# B&R Automation Studio project AAU12Segmenter (part 9)

#### mxA_Main.st - not listed in the package file held
```iecst
PROGRAM _INIT

	FOR i:=0 TO 5 DO
		KUKAs[i].AxisGroupIdx := i + 1;
		KUKAs[i].gripperAction.whitePin := ADR(gripperWhitePins[i]);
		KUKAs[i].gripperAction.blackPin := ADR(gripperBlackPins[i]);
		KUKAs[i].gripperAction.action := OPEN;
		KUKAs[i].gripperAction();
		KUKAs[i].cm.state := 0;
		KUKAs[i].startState := 0;
	END_FOR

	KUKAs[0].eeType := COVER_EE;
	KUKAs[1].eeType := DRILL_EE;
	KUKAs[2].eeType := PCB_EE;
	KUKAs[3].eeType := FUSE_EE;
	KUKAs[4].eeType := COVER_EE;
	KUKAs[5].eeType := COVER_EE;

END_PROGRAM

PROGRAM _CYCLIC

	// Loop through each robot for configurations
	FOR i := 0 TO 5 DO

		////////// Temporary skip until problem with library for Kuka KR4 is solved///////////
		IF i = 0 OR i = 5 THEN

			RETURN;

		END_IF

		/////////////////////////////////////////////////////
		// Logic to transform USINT (Input) to BYTE (FUBS) //
		/////////////////////////////////////////////////////

		brsmemcpy(ADR(KRC_Input[0]),ADR(InputVariables[i,0]), 254);

		/////////////////////////////////////////////////////
		// KRC_ReadAxisGroup has to be called at the Begin //
		// of the Cyclic Task to get all the Information   //
		// From the KRC from all KUKAs					   //
		/////////////////////////////////////////////////////

		KUKAs[i].start.KRC_ReadAxisGroup.KRC4_Input 			:= ADR(KRC_Input);
		KUKAs[i].start.KRC_ReadAxisGroup.AxisGroupIdx 			:= KUKAs[i].AxisGroupIdx;
		KUKAs[i].start.KRC_ReadAxisGroup.KRC_AxisGroupRefArr 	:= ADR(AxisRef);

		KUKAs[i].start.KRC_ReadAxisGroup();

		/////////////////////////////////////////////////////
		// Call User functions                             //
		/////////////////////////////////////////////////////

		pKuka ACCESS ADR(KUKAs[i]);
		cm ACCESS ADR(KUKAs[i].cm);

		// mxA_Start contains FB calls associated with initialization of the robots and diagnosis
		mxA_Start;

		//mxA_JointMovement;
		//mxA_LinearMovement;
		//mxA_ErrorMessage;

		CASE i OF
			1:
				mxA_KUKA1;

			2:
				mxA_KUKA2;

			3:
				mxA_KUKA3;

			4:
				mxA_KUKA4;

			5:
				mxA_KUKA5;

			6:
				mxA_KUKA6;

		END_CASE

		//mxA_KUKA6;

		/////////////////////////////////////////////////////
		// FunctionBlock to write the Output on the Struct //
		/////////////////////////////////////////////////////

		KUKAs[i].start.KRC_WriteAxisGroup.AxisGroupIdx			:= KUKAs[i].AxisGroupIdx;
		KUKAs[i].start.KRC_WriteAxisGroup.KRC_AxisGroupRefArr 	:= ADR(AxisRef);
		KUKAs[i].start.KRC_WriteAxisGroup.KRC4_Output 			:= ADR(KRC_Output);

		KUKAs[i].start.KRC_WriteAxisGroup();

		/////////////////////////////////////////////////////
		// Logic to transform BYTE (FUBS) to USINT (Input) //
		/////////////////////////////////////////////////////
		brsmemcpy(ADR(OutputVariables[i,0]),ADR(KRC_Output[0]), 254);

	END_FOR

END_PROGRAM
```

#### mxA_Start.st - not listed in the package file held
```iecst
ACTION mxA_Start:

	CASE pKuka.startState OF

		0: // Configuring KUKA FBs once

			// Logic to call the KRC_Initialize
			pKuka.start.KRC_Initialize.AxisGroupIdx 				:= pKuka.AxisGroupIdx;
			pKuka.start.KRC_Initialize.KRC_AxisGroupRefArr 			:= ADR(AxisRef);

			// Logic to call the KRC_Error
			pKuka.start.KRC_Error.AxisGroupIdx 						:= pKuka.AxisGroupIdx;
			pKuka.start.KRC_Error.MessageReset 						:= FALSE; // REMEMBER TO CHANGE LATER
			pKuka.start.KRC_Error.KRC_AxisGroupRefArr				:= ADR(AxisRef);

			// Logic to call KRC_AutomaticExternal
			pKuka.start.KRC_AutomaticExternal.AxisGroupIdx 			:= pKuka.AxisGroupIdx;
			pKuka.start.KRC_AutomaticExternal.MOVE_ENABLE 			:= TRUE;
			pKuka.start.KRC_AutomaticExternal.DRIVES_OFF 			:= TRUE;
			pKuka.start.KRC_AutomaticExternal.KRC_AxisGroupRefArr	:= ADR(AxisRef);
			pKuka.start.KRC_AutomaticExternal.EXT_START 			:= FALSE; // Binded to Continue Prog in original program
			pKuka.start.KRC_AutomaticExternal.ENABLE_T1 			:= TRUE;
			pKuka.start.KRC_AutomaticExternal.ENABLE_EXT 			:= TRUE;

			// Logic for startup of robot
			pKuka.start.KRC_AutoStart.AxisGroupIdx 					:= pKuka.AxisGroupIdx;
			pKuka.start.KRC_AutoStart.KRC_AxisGroupRefArr 			:= ADR(AxisRef);
			pKuka.start.KRC_AutoStart.ExecuteReset 					:= FALSE; // REMEMBER TO CHANGE LATER

			// Logic to set override for robot velocity
			pKuka.start.KRC_SetOverride.AxisGroupIdx 				:= pKuka.AxisGroupIdx;
			pKuka.start.KRC_SetOverride.KRC_AxisGroupRefArr 		:= ADR(AxisRef);
			pKuka.start.KRC_SetOverride.Override 					:= 10; // REMEMBER TO CHANGE LATER

			// Logic to set
			pKuka.start.KRC_Abort.AxisGroupIdx 						:= pKuka.AxisGroupIdx;
			pKuka.start.KRC_Abort.KRC_AxisGroupRefArr				:= ADR(AxisRef);
			pKuka.start.KRC_Abort.ExecuteCmd						:= FALSE;  /// Used to be set by HMI - Remember to incorporate it later

			// Logic to set KRC_Diag
			pKuka.start.KRC_Diag.AxisGroupIdx 						:= pKuka.AxisGroupIdx;
			pKuka.start.KRC_Diag.KRC_AxisGroupRefArr 				:= ADR(AxisRef);
			pKuka.start.KRC_Diag.ShowTrace 							:= FALSE;

			pKuka.startState  := 1;

		1: // Wait for P, S and EXT
			IF pKuka.status.P_ AND pKuka.status.S_ AND pKuka.status.EXT_ THEN

				pKuka.startState  := 2;

			END_IF

		2: // Reset KRC errors and autostart
			pKuka.start.KRC_Error.MessageReset := TRUE;
			pKuka.start.KRC_AutoStart.ExecuteReset := TRUE;

			IF pKuka.status.R_ AND pKuka.status.I_ THEN

				pKuka.start.KRC_Error.MessageReset := FALSE;
				pKuka.start.KRC_AutoStart.ExecuteReset := FALSE;
				pKuka.startState  := 3;

			END_IF

		3: // Check if any error occurred
			IF 	NOT pKuka.status.P_ OR
				NOT pKuka.status.S_ OR
				NOT pKuka.status.EXT_ OR
				NOT pKuka.status.R_ OR
				NOT pKuka.status.I_ THEN

				pKuka.startState  := 1;

			END_IF

	END_CASE

	// Logic to call the KRC_Initialize
	// KRC_Initialize gives back the Status OF the like, online, Initialized,.......
	pKuka.start.KRC_Initialize();

	// Logic to call the KRC_Error.
	// KRC_Error gives back the Status OF the Robot like, online, Initialized,.......
	pKuka.start.KRC_Error();

	// KRC_AutomaticExternal allows to control the Robot with the PLC
	pKuka.start.KRC_AutomaticExternal();

	//Function Block for StartUp of Robot
	pKuka.start.KRC_AutoStart();

	// KRC_SetOverride used to set the Override for the Robot Velocity
	pKuka.start.KRC_SetOverride();

	// KRC_Abort cancels all active and buffered statements and motions
	pKuka.start.KRC_Abort();

	// KRC_Diag gives back some information about the axis and robot
	pKuka.start.KRC_Diag();

	//Checking status of KRC and PLC for creating the signals for the HMI
	IF pKuka.start.KRC_Diag.ProconosCyc_Act = -1 OR pKuka.start.KRC_Error.NoHeartbeatPCOS THEN
		pKuka.status.P_ := FALSE;
	ELSE
		pKuka.status.P_ := TRUE;
	END_IF

	IF pKuka.start.KRC_Diag.SubmitCyc_Act = -1 OR pKuka.start.KRC_Error.NoHeartbeatKRC THEN
		pKuka.status.S_ := FALSE;
	ELSE
		pKuka.status.S_ := TRUE;
	END_IF

	IF pKuka.start.KRC_AutomaticExternal.EXT THEN
		pKuka.status.EXT_ := TRUE;
	ELSE
		pKuka.status.EXT_ := FALSE;
	END_IF

	IF NOT pKuka.start.KRC_Error.DrivesNotReady AND pKuka.start.KRC_AutomaticExternal.RC_RDY1 THEN
		pKuka.status.I_ := TRUE;
	ELSE
		pKuka.status.I_ := FALSE;
	END_IF

	IF pKuka.start.KRC_AutoStart.DispActive THEN
		pKuka.status.R_	:= TRUE;
	ELSE
		pKuka.status.R_	:= FALSE;
	END_IF

END_ACTION
```

#### RobotHandling.st - not listed in the package file held
```iecst
ACTION RobotHandling:
	CASE cm.state OF

		1000:
			IF robotExecute[i] THEN
				cm.description := 'Move to pickup point with relative linear movement';
				robotBusy[i] := TRUE;
				pKuka.convert.ValuesToCOORDSYS.IPO_Mode := 1; // #TOOL
				pKuka.convert.ValuesToCOORDSYS();

				pKuka.motion.KRC_MoveLinearRelative.CoordinateSystem := pKuka.convert.ValuesToCOORDSYS.COORDSYS;

				pKuka.tempPosition.X := pKuka.tempPosition.Y := pKuka.tempPosition.Z := pKuka.tempPosition.A := pKuka.tempPosition.B := pKuka.tempPosition.C
				:= 0;
				pKuka.tempPosition.Z := -relativeDistance;
				// Status and turn is already set from moving to approach point

				pKuka.motion.KRC_MoveLinearRelative.Position := pKuka.tempPosition;

				pKuka.motion.KRC_MoveLinearRelative.ExecuteCmd := TRUE;
				IF pKuka.motion.KRC_MoveLinearRelative.Done THEN
					pKuka.motion.KRC_MoveLinearRelative.ExecuteCmd := FALSE;
					cm.state := 1010;
				END_IF
			END_IF

		1010:
			cm.description := 'Close gripper and wait a little before moving to ensure proper grip';

			pKuka.gripperAction.action := CLOSE;

			pKuka.TON.PT := REAL_TO_TIME(gripperWaitTime); // in ms
			pKuka.TON.IN := TRUE;
			IF pKuka.TON.Q THEN
				pKuka.TON.IN := FALSE;
				cm.state := 1020;
			END_IF

		1020:
			cm.description := 'Move back to approach point with relative linear movement';

			pKuka.tempPosition.X := pKuka.tempPosition.Y := pKuka.tempPosition.Z := pKuka.tempPosition.A := pKuka.tempPosition.B := pKuka.tempPosition.C
			:= 0;
			pKuka.tempPosition.Z := relativeDistance;
			// Status and turn is already set from moving to approach point

			pKuka.motion.KRC_MoveLinearRelative.Position := pKuka.tempPosition;

			pKuka.motion.KRC_MoveLinearRelative.ExecuteCmd := TRUE;
			IF pKuka.motion.KRC_MoveLinearRelative.Done THEN
				pKuka.motion.KRC_MoveLinearRelative.ExecuteCmd := FALSE;
				cm.state := 1030;
			END_IF

		1030:
			cm.description := 'Move to approach point of magazine with absolute direct movement';

			pKuka.convert.ValuesToPosition.posType := APPROACH_MAGAZINE;
			pKuka.convert.ValuesToPosition();

			pKuka.convert.ValuesToCOORDSYS.Base := pKuka.convert.ValuesToPosition.baseNo; // Magazine frame
			pKuka.convert.ValuesToCOORDSYS.IPO_Mode := 0; // #BASE
			pKuka.convert.ValuesToCOORDSYS();

			pKuka.tempPosition := pKuka.convert.ValuesToPosition.outputPos;

			pKuka.motion.KRC_MoveDirectAbsolute.CoordinateSystem := pKuka.convert.ValuesToCOORDSYS.COORDSYS;
			pKuka.motion.KRC_MoveDirectAbsolute.Position := pKuka.tempPosition;

			pKuka.motion.KRC_MoveDirectAbsolute.ExecuteCmd := TRUE;
			IF pKuka.motion.KRC_MoveDirectAbsolute.Done THEN
				pKuka.motion.KRC_MoveDirectAbsolute.ExecuteCmd := FALSE;
				cm.state := 1040;
			END_IF

		1040:
			cm.description := 'Define order-specific approach point at magazine';

			pKuka.convert.ValuesToPosition.posType := APPROACH_MAGAZINE;
			pKuka.convert.ValuesToPosition();

			pKuka.tempPosition := pKuka.convert.ValuesToPosition.outputPos;

			CASE pKuka.axisGroupIdx OF
				6:
					// Determine the stack the manipulator should go to depending on the ID of the order
					FOR k := 0 TO (unloadSizeX*unloadSizeY - 1) DO
						xIdxTemp := k MOD unloadSizeX;
						yIdxTemp := REAL_TO_INT(brmfloor(k / unloadSizeX));

						// If the ID already has a stack
						IF idAtStack[xIdxTemp, yIdxTemp] = orderSpec[i] THEN
							// If an non-taken stack was selected, reset it
							IF (xIdx <> -1 OR yIdx <> -1) THEN
								idAtStack[xIdx, yIdx] := -1;
							END_IF
							xIdx := xIdxTemp;
							yIdx := yIdxTemp;
							EXIT;
						END_IF

						IF (xIdx = -1 OR yIdx = -1) AND (idAtStack[xIdxTemp, yIdxTemp] = -1 AND stackCounter[xIdxTemp, yIdxTemp] + orderAmount <= unloadSizeZ) THEN
							xIdx := xIdxTemp;
							yIdx := yIdxTemp;
							idAtStack[xIdx, yIdx] := orderSpec[i];
						END_IF

					END_FOR

					// Determine the position from x- and y-index
					pKuka.tempPosition.X := pKuka.tempPosition.X + xIdx * 120;
					pKuka.tempPosition.Y := pKuka.tempPosition.Y - yIdx * 80;

					// Reset parameters and increment counters
					orderCounter[xIdx, yIdx] := orderCounter[xIdx, yIdx] + 1;
					stackCounter[xIdx, yIdx] := stackCounter[xIdx, yIdx] + 1;
					IF orderCounter[xIdx, yIdx] = orderAmount THEN
						idAtStack[xIdx, yIdx] := -1;
						orderCounter[xIdx, yIdx] := 0;
					END_IF
					xIdx := yIdx := -1;

			END_CASE

			cm.state := 1050;

		1050:
			cm.description := 'Move to order-specific approach point at magazine';
			pKuka.convert.ValuesToCOORDSYS.IPO_Mode := 0; // #BASE
			pKuka.convert.ValuesToCOORDSYS();

			pKuka.motion.KRC_MoveDirectAbsolute.CoordinateSystem := pKuka.convert.ValuesToCOORDSYS.COORDSYS;

			pKuka.motion.KRC_MoveDirectAbsolute.Position := pKuka.tempPosition;

			pKuka.motion.KRC_MoveDirectAbsolute.ExecuteCmd := TRUE;
			IF pKuka.motion.KRC_MoveDirectAbsolute.Done THEN
				pKuka.motion.KRC_MoveDirectAbsolute.ExecuteCmd := FALSE;
				cm.state := 1060;
			END_IF

		1060:
			cm.description := 'Move to place point at magazine with relative movement';

			pKuka.convert.ValuesToCOORDSYS.IPO_Mode := 1; // #TOOL
			pKuka.convert.ValuesToCOORDSYS();

			pKuka.motion.KRC_MoveLinearRelative.CoordinateSystem := pKuka.convert.ValuesToCOORDSYS.COORDSYS;

			pKuka.tempPosition.X := pKuka.tempPosition.Y := pKuka.tempPosition.A := pKuka.tempPosition.B := pKuka.tempPosition.C
			:= 0;
			pKuka.tempPosition.Z := -(pKuka.tempPosition.Z - (unloadSizeZ - stackCounter[xIdx,yIdx])* 21);
			// Status and turn is already set from moving to approach point

			pKuka.motion.KRC_MoveLinearRelative.Position := pKuka.tempPosition;

			pKuka.motion.KRC_MoveLinearRelative.ExecuteCmd := TRUE;
			IF pKuka.motion.KRC_MoveLinearRelative.Done THEN
				pKuka.motion.KRC_MoveLinearRelative.ExecuteCmd := FALSE;
				cm.state := 1070;
			END_IF

		1070:
			cm.description := 'Open gripper and wait a little before moving to ensure proper grip';

			pKuka.gripperAction.action := OPEN;

			pKuka.TON.PT := REAL_TO_TIME(gripperWaitTime); // in ms
			pKuka.TON.IN := TRUE;
			IF pKuka.TON.Q THEN
				pKuka.TON.IN := FALSE;
				cm.state := 1080;
			END_IF

		1080:
			cm.description := 'Move to place point at magazine with relative movement';

			pKuka.convert.ValuesToCOORDSYS.IPO_Mode := 1; // #TOOL
			pKuka.convert.ValuesToCOORDSYS();

			pKuka.motion.KRC_MoveLinearRelative.CoordinateSystem := pKuka.convert.ValuesToCOORDSYS.COORDSYS;

			pKuka.tempPosition.X := pKuka.tempPosition.Y := pKuka.tempPosition.A := pKuka.tempPosition.B := pKuka.tempPosition.C
			:= 0;
			pKuka.tempPosition.Z := (pKuka.tempPosition.Z - (unloadSizeZ - stackCounter[xIdx,yIdx])* 21);
			// Status and turn is already set from moving to approach point

			pKuka.motion.KRC_MoveLinearRelative.Position := pKuka.tempPosition;

			pKuka.motion.KRC_MoveLinearRelative.ExecuteCmd := TRUE;
			IF pKuka.motion.KRC_MoveLinearRelative.Done THEN
				pKuka.motion.KRC_MoveLinearRelative.ExecuteCmd := FALSE;
				robotDone[i] := TRUE;
				cm.state := 1090;
			END_IF

		1090:
			cm.description := 'Move back to home position';
			RobotHoming;

	END_CASE
END_ACTION
```

#### RobotProgram.st - not listed in the package file held
```iecst
ACTION RobotProgram:

	//JointMovement;
	//LinearMovement;
	//ErrorMessage;

	CASE pKuka.axisGroupIdx OF
		1:
			KUKABottomCover;

		2:
			//KUKADrilling;
			LinearMovement;

		3:
			KUKAPcb;

		4:
			KUKAFuse;

		5:
			KUKATopCover;

		6:
			KUKAUnloading;

	END_CASE

END_ACTION
```

### Program Logical/Modules/KUKA/Services/HMI/HMI (IEC)

#### drawConfigShuttles.st
```iecst
ACTION drawConfigShuttles:
	IF shuttleStartPosSvg OR init THEN
		IF i = 0 THEN
		showConfigShuttles := '';
		tmpString := showMotorSegments;
		brdkStrRemove(ADR(tmpString),-1,1);
		brdkStrCat(ADR(showConfigShuttles), ADR(tmpString));
		brdkStrCat(ADR(showConfigShuttles), ADR(','));
		END_IF

		brdkStrCat(ADR(showConfigShuttles), ADR('{"select":"#rect'));

		tmpString := USINT_TO_STRING(i+1);
		brdkStrCat(ADR(showConfigShuttles), ADR(tmpString));
		brdkStrCat(ADR(showConfigShuttles), ADR('","display":'));
		IF (nrOfShuttlesHMI >= (i+1)) THEN
			brdkStrCat(ADR(showConfigShuttles), ADR('true'));
		ELSE
			brdkStrCat(ADR(showConfigShuttles), ADR('false'));
		END_IF

		brdkStrCat(ADR(showConfigShuttles), ADR(',"translate":['));

		tmpCalc := (pShuttleStartupInfo.initXPos*1000)-60;
		tmpString := REAL_TO_STRING(tmpCalc);
		brdkStrCat(ADR(showConfigShuttles), ADR(tmpString));
		brdkStrCat(ADR(showConfigShuttles), ADR(','));

		tmpCalc := 1200 - (pShuttleStartupInfo.initYPos*1000) - 60;
		tmpString := REAL_TO_STRING(tmpCalc);
		brdkStrCat(ADR(showConfigShuttles), ADR(tmpString));

		IF i = NUM_SHUTTLES THEN
			brdkStrCat(ADR(showConfigShuttles), ADR(']}]'));
		ELSE
		brdkStrCat(ADR(showConfigShuttles), ADR(']},'));
		END_IF
	END_IF

END_ACTION
```

### Types.typ
```iecst
TYPE
	lightControlCenter_typ : 	STRUCT
		visionProgram : BOOL;
		shuttlePrecision : BOOL;
		weightProgram : BOOL;
		gameProgram : BOOL;
		linkProgram : BOOL;
		coneveyorMovementProgram : BOOL;
		intelligentMovementProgram : BOOL;
		demoProgram : BOOL;
	END_STRUCT;
END_TYPE
```

### Program Logical/Modules/KUKA/Services/HMI/Vision/Vi_main

#### Main.st
```iecst
// --------------------------------------------------------------------------------------------------------------------
// General vision task. This is a support task for the mappView visualization. The following functions are implemneted
// - Disable mappView functions when camera is not ready, available
// - Load image on main page when camera has finished inspection
// - Transfer parameters after vision setup
// - Draw crosshairs into image on the main page
// Version 2.x (Check revision history for details)
// --------------------------------------------------------------------------------------------------------------------
PROGRAM _INIT
	// -----------------------------------------------------------------------------------------------------------
	// Map global structure to local reference
	VisionSensor ACCESS ADR(gVisionSensor[visSelectedSensor]);
	Blob ACCESS ADR(tmpBlob);
	CodeReader ACCESS ADR(tmpCodeReader);
	Match ACCESS ADR(tmpMatch);
	MT ACCESS ADR(tmpMT);
	OCR ACCESS ADR(tmpOCR);

	// -----------------------------------------------------------------------------------------------------------
	// Preload code types
	FOR i := 0 TO MAX_NUM_CODETYPES DO
		IF CodeTypes[i] <> '' THEN
			brsstrcat(ADR(visCodeTypePresentDropDownValues[i]), ADR('{"value":"'));
			brsitoa(i, ADR(tmpStr1));
			brsstrcat(ADR(visCodeTypePresentDropDownValues[i]), ADR(tmpStr1));
			brsstrcat(ADR(visCodeTypePresentDropDownValues[i]), ADR('","text":"'));
			brsstrcat(ADR(visCodeTypePresentDropDownValues[i]), ADR(CodeTypes[i]));
			brsstrcat(ADR(visCodeTypePresentDropDownValues[i]), ADR('"}'));
		END_IF
	END_FOR

	// -----------------------------------------------------------------------------------------------------------
	visTableNo;
	InitialSearchSensor := TRUE;
END_PROGRAM

// -----------------------------------------------------------------------------------------------------------
// Cyclic part
// -----------------------------------------------------------------------------------------------------------
PROGRAM _CYCLIC
// -----------------------------------------------------------------------------------------------------------
// Part 1: Things to be done for every camera/sensor
// -----------------------------------------------------------------------------------------------------------
	FOR idx := 1 TO MAX_NUM_CAMS DO
		// -----------------------------------------------------------------------------------------------------------
		// Display camera status in hex - documenation is also in hex
		// -----------------------------------------------------------------------------------------------------------
		IF gVisionSensor[idx].DAT.Status = 0 THEN // Display only a single 0
			gVisionSensor[idx].DAT.StatusText := '0';
		ELSIF gVisionSensor[idx].DAT.Status = 16#00000001 THEN
			gVisionSensor[idx].DAT.StatusText := 'Image acquisition';
		ELSIF gVisionSensor[idx].DAT.Status = 16#00000002 THEN
			gVisionSensor[idx].DAT.StatusText := 'Waiting trigger';
		ELSIF gVisionSensor[idx].DAT.Status = 16#00000010 THEN
			gVisionSensor[idx].DAT.StatusText := 'Searching settings';
		ELSIF gVisionSensor[idx].DAT.Status = 16#00000080 THEN
			gVisionSensor[idx].DAT.StatusText := 'Setting focus';
		ELSIF gVisionSensor[idx].DAT.Status = 16#00000090 THEN
			gVisionSensor[idx].DAT.StatusText := 'Searching settings';
		ELSIF gVisionSensor[idx].DAT.Status = 16#00000800 THEN
			gVisionSensor[idx].DAT.StatusText := 'Cam CPU not ready';
		ELSIF gVisionSensor[idx].DAT.Status = 16#00001000 THEN
			gVisionSensor[idx].DAT.StatusText := 'Cam sensor not ready';
		ELSIF gVisionSensor[idx].DAT.Status = 16#02000000 THEN
			gVisionSensor[idx].DAT.StatusText := 'OS check/update';
		ELSIF gVisionSensor[idx].DAT.Status = 16#80000000 THEN
			gVisionSensor[idx].DAT.StatusText := 'Vision cockpit active';
		ELSE // Display the status in hex format 0x02000800
			gVisionSensor[idx].DAT.StatusText := '';
			FOR i := 0 TO 28 BY 4 DO
				gVisionSensor[idx].DAT.StatusText := CONCAT(MID(HexTab, 1, LIMIT(1, UDINT_TO_INT((SHR(gVisionSensor[idx].DAT.Status, i) AND 16#0000000F) + 1), 16)), gVisionSensor[idx].DAT.StatusText);
			END_FOR
			gVisionSensor[idx].DAT.StatusText := CONCAT('0x', gVisionSensor[idx].DAT.StatusText);
		END_IF

		// -----------------------------------------------------------------------------------------------------------
		// Check if vision cockpit is open
		// -----------------------------------------------------------------------------------------------------------
		gVisionSensor[idx].DAT.CockpitIsActive := (gVisionSensor[idx].DAT.Status AND 16#8000_0000) > 0;

		// -----------------------------------------------------------------------------------------------------------
		// Auto setup handling
		// -----------------------------------------------------------------------------------------------------------
		IF(gVisionSensor[idx].CMD.AutoSetupStartStop AND gVisionSensor[idx].DAT.Status <> 0) THEN
			AutoSetupRunning[idx] := TRUE;
		ELSIF NOT gVisionSensor[idx].CMD.AutoSetupStartStop THEN
			AutoSetupRunning[idx] := FALSE;
		END_IF
		IF(gVisionSensor[idx].CMD.AutoSetupStartStop AND gVisionSensor[idx].DAT.Status = 0 AND AutoSetupRunning[idx]) THEN // Setup successfully finished
			gVisionSensor[idx].DAT.Gain					:= gVisionSensor[idx].DAT.AutoSetupGain;
			gVisionSensor[idx].DAT.Focus				:= gVisionSensor[idx].DAT.AutoSetupFocus;
			gVisionSensor[idx].DAT.Exposure				:= gVisionSensor[idx].DAT.AutoSetupExposure;
			gVisionSensor[idx].CMD.AutoSetupStartStop	:= FALSE;
			AutoSetupRunning[idx]						:= FALSE;
			TON_DelayAfterAutoSetup.IN					:= TRUE;
		END_IF
		TON_DelayAfterAutoSetup(PT := T#50ms);
		IF TON_DelayAfterAutoSetup.Q THEN // After the camera tells it is ready, we need to wait still at least ca 20ms, otherwise it does not accept the trigger
			TON_DelayAfterAutoSetup.IN := FALSE;
			IF gVisionSensor[idx].HW.Ready AND NOT gVisionSensor[idx].DAT.ImageProcessingActive THEN
				gVisionSensor[idx].DAT.NettimeDelay	:= NettimeCurrent_us + NETTIME_DEFAULT_DELAY;
				gVisionSensor[idx].CMD.ImageTrigger	:= TRUE;
				gVisionSensor[idx].DAT.Active			:= TRUE;
			END_IF
		END_IF

		// -----------------------------------------------------------------------------------------------------------
		// Reset image trigger, reload web page and store image when process is finished
		// -----------------------------------------------------------------------------------------------------------
		IF ((gVisionSensor[idx].DAT.AcquisitionCompletedCnt <> AcquisitionCompletedCntOld[idx] OR gVisionSensor[idx].DAT.AcquisitionFailedCnt <> AcquisitionFailedCntOld[idx]) AND NOT gVisionSensor[idx].DAT.ImageProcessingActive AND gVisionSensor[idx].HW.Ready) THEN
			AcquisitionCompletedCntOld[idx]			:= gVisionSensor[idx].DAT.AcquisitionCompletedCnt;
			AcquisitionFailedCntOld[idx]			:= gVisionSensor[idx].DAT.AcquisitionFailedCnt;
			gVisionSensor[idx].CMD.ImageTrigger		:= FALSE;
			gVisionSensor[idx].DAT.Active			:= FALSE;
			// Store image to flash card, only for the actual selected camera
			IF idx = visSelectedSensor THEN
				IF visAutoArchiv AND NOT DisableAutoArchiv THEN
					gVisionImage.CMD.SaveImageOnPLC := TRUE;
				END_IF
				IF NOT visRepetitiveMode THEN
					DisableAutoArchiv := FALSE;
				END_IF
			END_IF
		END_IF

		// -----------------------------------------------------------------------------------------------------------
		// Reset trigger when timed out
		// -----------------------------------------------------------------------------------------------------------
		IF gVisionSensor[idx].CMD.ImageTrigger THEN
			TriggerTimeout[idx].IN := TRUE;
			TriggerTimeout[idx].PT := REAL_TO_TIME(gVisionSensor[idx].DAT.Timeout * 1.25);
			IF TriggerTimeout[idx].Q THEN
				gVisionSensor[idx].CMD.ImageTrigger			:= FALSE;
				gVisionSensor[idx].CMD.ImageTriggerReset	:= TRUE;
				gVisionSensor[idx].DAT.Active				:= FALSE;
			END_IF
		ELSE
			TriggerTimeout[idx].IN := FALSE;
			gVisionSensor[idx].CMD.ImageTriggerReset := FALSE;
		END_IF
		TriggerTimeout[idx]();
	END_FOR

// -----------------------------------------------------------------------------------------------------------
// Part 2: Things to be done for the actual selected camera / visualization related things
// -----------------------------------------------------------------------------------------------------------
	// -----------------------------------------------------------------------------------------------------------
	// Select first available camera after reboot
	// -----------------------------------------------------------------------------------------------------------
	IF InitialSearchSensor THEN
		FOR i := 1 TO MAX_NUM_CAMS DO
			IF gVisionSensor[i].HW.Connected THEN
				visSelectedSensor := i;
				InitialSearchSensor := FALSE;
				EXIT;
			END_IF
		END_FOR
		visVaListRefresh := TRUE;
	END_IF

	// -----------------------------------------------------------------------------------------------------------
	// Map global structure to local reference for mappView
	// -----------------------------------------------------------------------------------------------------------
	// Make sure we dont exceed array limit
	IF(visSelectedSensor > MAX_NUM_CAMS) THEN
		visSelectedSensor := 1;
	END_IF
	IF(visSelectedSensor < 1) THEN
		visSelectedSensor := MAX_NUM_CAMS;
	END_IF
	// -----------------------------------------------------------------------------------------------------------
	// Assign pointers
	VisionSensor ACCESS ADR(gVisionSensor[visSelectedSensor]);
	IF(VisionSensor.CFG.DataStructure <> 0) THEN
		CASE VisionSensor.CFG.VisionFunction OF
			enumBlob:			Blob ACCESS VisionSensor.CFG.DataStructure;
			enumCoderReader:	CodeReader ACCESS VisionSensor.CFG.DataStructure;
			enumMatch:			Match ACCESS VisionSensor.CFG.DataStructure;
			enumMeasurement:	MT ACCESS VisionSensor.CFG.DataStructure;
			enumOCR:			OCR ACCESS VisionSensor.CFG.DataStructure;
		END_CASE
	ELSE
		RETURN;
	END_IF

	// -----------------------------------------------------------------------------------------------------------
	// Display camera status
	// -----------------------------------------------------------------------------------------------------------
	visCameraStatus := VisionSensor.DAT.StatusText;

	// -----------------------------------------------------------------------------------------------------------
	// Code Reader - selected/detected types
	// -----------------------------------------------------------------------------------------------------------
	IF VisionSensor.CFG.VisionFunction = enumCoderReader THEN
		IF(visSelectedCodeTypeToPLC <> '') THEN
			CodeReader.CodeType := UDINT_TO_USINT(brsatoi(ADR(visSelectedCodeTypeToPLC)));
			visSelectedCodeTypeToPLC := '';
		END_IF
		brsitoa(CodeReader.CodeType, ADR(visSelectedCodeTypeFromPLC));
		FOR i := 1 TO MAX_NUM_RESULTS DO
			IF CodeReader.BarcodeType[i] <> 0 THEN
				brsstrcpy(ADR(visSelectedCodeTypeDetected[i]), ADR(CodeTypes[LIMIT(0, CodeReader.BarcodeType[i], MAX_NUM_CODETYPES)]));
			ELSE
				brsstrcpy(ADR(visSelectedCodeTypeDetected[i]), ADR(''));
			END_IF
		END_FOR
	END_IF

	// -----------------------------------------------------------------------------------------------------------
	// Translate flash color and segments from mappView to IO mapping
	// -----------------------------------------------------------------------------------------------------------
	// Hint: Normally copy from recipe (VisionSensor) to visu. Only in case of a change in the visu copy to recipe
	IF visSelectedFlashColor <> visSelectedFlashColorOld THEN // The flash color was changed in the mappView visualization
		VisionSensor.DAT.FlashColor := UDINT_TO_USINT(brsatoi(ADR(visSelectedFlashColor)));
	ELSE
		brsitoa(VisionSensor.DAT.FlashColor, ADR(visSelectedFlashColor));
	END_IF
	visSelectedFlashColorOld := visSelectedFlashColor;
	IF brsmemcmp(ADR(visSelectedFlashSegment), ADR(visSelectedFlashSegmentOld), SIZEOF(visSelectedFlashSegment)) <> 0 THEN // The flash segments was changed in the mappView visualization
		VisionSensor.DAT.FlashSegment := SHL(visSelectedFlashSegment[0], 0) OR SHL(visSelectedFlashSegment[1], 1) OR SHL(visSelectedFlashSegment[2], 2) OR SHL(visSelectedFlashSegment[3], 3);
	ELSE
		visSelectedFlashSegment[0] := VisionSensor.DAT.FlashSegment.0;
		visSelectedFlashSegment[1] := VisionSensor.DAT.FlashSegment.1;
		visSelectedFlashSegment[2] := VisionSensor.DAT.FlashSegment.2;
		visSelectedFlashSegment[3] := VisionSensor.DAT.FlashSegment.3;
	END_IF
	visSelectedFlashSegmentOld := visSelectedFlashSegment;

	// -----------------------------------------------------------------------------------------------------------
	// Disable command buttons when camera is disconnected, not ready, processing an image or vision cockpit is open
	// -----------------------------------------------------------------------------------------------------------
	IF(NOT VisionSensor.HW.Connected OR NOT VisionSensor.HW.Ready OR VisionSensor.DAT.ImageProcessingActive OR VisionSensor.DAT.CockpitIsActive) THEN
		visEnableCommand := FALSE;
	ELSE
		visEnableCommand := TRUE;
	END_IF

	// -----------------------------------------------------------------------------------------------------------
	// Disable setup buttons when camera is disconnected, processing an image or not ready
	// -----------------------------------------------------------------------------------------------------------
	IF(NOT VisionSensor.HW.Connected OR NOT (VisionSensor.HW.Ready OR AutoSetupRunning[visSelectedSensor]) OR VisionSensor.DAT.ImageProcessingActive) THEN
		visEnableSetup := FALSE;
	ELSE
		visEnableSetup := TRUE;
	END_IF

	// -----------------------------------------------------------------------------------------------------------
	// Fire trigger for camera image
	// -----------------------------------------------------------------------------------------------------------
	IF((visImageTrigger OR EDGEPOS(visEnableVision)) AND VisionSensor.HW.Ready AND NOT VisionSensor.DAT.ImageProcessingActive) THEN
		// Add default delay and fire trigger
		VisionSensor.DAT.NettimeDelay	:= NettimeCurrent_us + NETTIME_DEFAULT_DELAY;
		VisionSensor.CMD.ImageTrigger	:= TRUE;
		visImageTrigger					:= FALSE;
		VisionSensor.DAT.Active			:= TRUE;
	END_IF

	// -----------------------------------------------------------------------------------------------------------
	// Repetitive mode
	// -----------------------------------------------------------------------------------------------------------
	visEnableRepetitive := visEnableCommand OR visRepetitiveMode; // Enable of the repetitive mode button. Don't disable while repetitive mode is active
	IF visRepetitiveMode THEN
		RepetitiveModeTimer.IN := TRUE;
		IF RepetitiveModeTimer.Q THEN
			IF VisionSensor.HW.Ready AND NOT VisionSensor.DAT.ImageProcessingActive THEN
				RepetitiveModeTimer.IN := FALSE;
				VisionSensor.DAT.NettimeDelay := NettimeCurrent_us + NETTIME_DEFAULT_DELAY;
				VisionSensor.CMD.ImageTrigger := TRUE;
			END_IF
		END_IF
		DisableAutoArchiv := TRUE;
	ELSE
		RepetitiveModeTimer.IN := TRUE;
	END_IF
	RepetitiveModeTimer(PT := T#200ms);
	VisionSensor.DAT.Enable := visEnableVision AND NOT visRepetitiveMode;

	// -----------------------------------------------------------------------------------------------------------
	// Get list of vision applications and components
	// -----------------------------------------------------------------------------------------------------------
	IF (visVaListRefresh) THEN
		VaGetList_01(Enable := TRUE);
		VisionSensor.FCT.Status := ERR_FUB_BUSY;
		IF VaGetList_01.Status <> ERR_FUB_BUSY THEN
			// Convert vision application list to mappView format
			IF VaGetList_01.Status = ERR_OK THEN
				IF VaGetList_01.VaApplicationCnt > 0 AND VaGetList_01.VaApplicationCnt < MAX_IDX_VA_LIST THEN
					FOR i:=0 TO VaGetList_01.VaApplicationCnt - 1 DO
						String2DataProvider(ADR(VaGetList_01.VaApplicationNames[i]), ADR(visVisionApplicationList[i]));
					END_FOR
				END_IF
				VisionSensor.FCT.Status := ERR_OK;
			ELSE // Error
				brsmemset(ADR(visVisionApplicationList), 0, SIZEOF(visVisionApplicationList));
				VisionSensor.FCT.Status := VaGetList_01.Status;
			END_IF
			// Reset function block
			VaGetList_01(Enable := FALSE);
			visVaListRefresh := FALSE;
		END_IF
	END_IF

	// -----------------------------------------------------------------------------------------------------------
	// Load vision application
	// -----------------------------------------------------------------------------------------------------------
	IF (VisionSensor.CMD.VaSwitchApplication) THEN
		ViBaseLoadApplication_01.MpLink	:= ADR(VisionSensor.CFG.ComponentLink);
		ViBaseLoadApplication_01.Name	:= ADR(VisionSensor.FCT.ApplicationName);
		VisionSensor.FCT.Status := ERR_FUB_BUSY;

		// -----------------------------------------------------------------------------------------------------------
		// OK
		IF (ViBaseLoadApplication_01.Done) THEN
			VisionSensor.FCT.Status := ERR_OK;
			VisionSensor.CMD.VaSwitchApplication := FALSE;
		// -----------------------------------------------------------------------------------------------------------
		// Error
		ELSIF (NOT ViBaseLoadApplication_01.Busy AND ViBaseLoadApplication_01.Error) THEN
			VisionSensor.FCT.Status := ViBaseLoadApplication_01.StatusID;
			VisionSensor.CMD.VaSwitchApplication := FALSE;
		END_IF
	END_IF
	ViBaseLoadApplication_01.Execute := VisionSensor.CMD.VaSwitchApplication;
	ViBaseLoadApplication_01();

	// -----------------------------------------------------------------------------------------------------------
	// Informations for Vi_image
	// -----------------------------------------------------------------------------------------------------------
	IF EDGENEG(VisionSensor.DAT.ImageProcessingActive) THEN
		gVisionImage.CMD.RefreshCrosshair := TRUE;
	END_IF
	gVisionImage.DAT.VisionDisabled := NOT visEnableVision;

	// -----------------------------------------------------------------------------------------------------------
	// Save diagnostic data
	// -----------------------------------------------------------------------------------------------------------
	IF (VisionSensor.CMD.SaveDiagData) THEN
		// Delete old file first
		FDelete.enable := VisionSensor.CMD.SaveDiagData AND NOT ViBaseSaveDiagData_01.Execute;
		FDelete.pDevice := ADR(DEVICE_NAME);
		FDelete.pName := ADR(VisionSensor.DIA.DiagName);
		IF (FDelete.status <> ERR_FUB_BUSY) THEN
			ViBaseSaveDiagData_01.Execute := TRUE;
		END_IF
		// Upload diagnostic information
		ViBaseSaveDiagData_01.MpLink := ADR(VisionSensor.CFG.ComponentLink);
		ViBaseSaveDiagData_01.DeviceName := ADR(DEVICE_NAME);
		ViBaseSaveDiagData_01.FileName := ADR(VisionSensor.DIA.DiagName);
		VisionSensor.DIA.Status := ERR_FUB_BUSY;

		// -----------------------------------------------------------------------------------------------------------
		// OK
		IF (ViBaseSaveDiagData_01.Done) THEN
			VisionSensor.DIA.Status := ERR_OK;
			ViBaseSaveDiagData_01.Execute := FALSE;
			VisionSensor.CMD.SaveDiagData := FALSE;
		// -----------------------------------------------------------------------------------------------------------
		// Error
		ELSIF (NOT ViBaseSaveDiagData_01.Busy AND ViBaseSaveDiagData_01.Error) THEN
			VisionSensor.DIA.Status := ViBaseSaveDiagData_01.StatusID;
			ViBaseSaveDiagData_01.Execute := FALSE;
			VisionSensor.CMD.SaveDiagData := FALSE;
		END_IF
	END_IF
	ViBaseSaveDiagData_01();
	FDelete();

END_PROGRAM
```

### Program Logical/Modules/KUKA/Services/HMI/Vision/Vision

#### Main.st
```iecst
// --------------------------------------------------------------------------------------------------------------------
// This task calculates the nettime depending on a drive velocity
// - This task must run at the same cycle as the Powerlink bus
// - Make sure that nettime is selected in the vision application (Image aquisition -> Aquisition configuration -> Trigger Source -> Trigger delay
// --------------------------------------------------------------------------------------------------------------------
PROGRAM _INIT
	(* Insert code here *)
	gVisionNettime.CMD.Activate					:= TRUE;
	gVisionNettime.CFG.AxisPeriod				:= 360; // Needs also to be set in the axis configuration
	gVisionNettime.CFG.AxisPositionTrigger		:= 0.180;
	gVisionNettime.CFG.AxisPositionDelay_Cycles	:= 1; 	// Number of PLK cycles which the axis position is old when it comes to this task (Time from encoder to now in this task)
	gVisionNettime.CFG.VisionPreTrigger_Cycles	:= 8; 	// Number of powerlink cycles the trigger has to be send ahead, 4 is a good value.

	mappView.maxSvgImageLength := SIZEOF(imageSvg);
	mappView.enable 		:= TRUE;
	mappView.cameraIp 		:= '192.168.200.8';
	mappView.getImageArray := FALSE;
	mappView.timeout 		:= 3000;

	//WHILE mappView.internal. = 0 DO
		mappView();
	//END_WHILE
	//	mappView.simulateConfig.appendNumber := TRUE;
//	mappView.simulateConfig.minNumber := 1;
//	mappView.simulateConfig.maxNumber := 3;
//	mappView.simulateConfig.autoIncrementNumber := TRUE;
//	mappView.simulateConfig.pDevice := ADR(this.simFileDevice);
//	mappView.simulateConfig.pFile := ADR(this.simFilename);
END_PROGRAM

PROGRAM _CYCLIC
	PowerlinkCycle_us			:= NettimeCurrent_us - NettimeLastCycle_us;
	NettimeLastCycle_us			:= NettimeCurrent_us;
	ShuttleYSpeed_ms			:= ((ShuttleYPos_m - ShuttleYPosOld_m[LAST_IDX_SH_POS_OLD]) / (LAST_IDX_SH_POS_OLD + 1) / MAX(PowerlinkCycle_us, 400) * 1000000)*(-1) ;
	brsmemmove(ADR(ShuttleYPosOld_m[1]), ADR(ShuttleYPosOld_m[0]), SIZEOF(ShuttleYPosOld_m) - SIZEOF(ShuttleYPosOld_m[0]));
	ShuttleYPosOld_m[0]			:= ShuttleYPos_m;

	IF gVisionNettime.CMD.Activate AND ShuttleYSpeed_ms > 0 THEN //AND gVisionNettime.DAT.AxisInVelocity AND gVisionNettime.DAT.AxisVelocity > 0 THEN
		AxisPositionNow			:= ShuttleYPos_m + (-1* ShuttleYSpeed_ms) * PowerlinkCycle_us * gVisionNettime.CFG.AxisPositionDelay_Cycles / 1000000; // When the MpAxis gives us the read position, it is old. So calculate the "now" position
		TriggerPosDelta			:= gVisionNettime.CFG.AxisPositionTrigger - AxisPositionNow;
		TriggerTimeDelta_us		:= LREAL_TO_DINT((TriggerPosDelta / ShuttleYSpeed_ms) * 1000000);
		// Wait for the moment that axis is in the send trigger window depend on delay by topology and the actual powerlink cycle
		IF (TriggerTimeDelta_us >= (gVisionNettime.CFG.VisionPreTrigger_Cycles)     * PowerlinkCycle_us)  AND
			(TriggerTimeDelta_us <= (gVisionNettime.CFG.VisionPreTrigger_Cycles + 1) * PowerlinkCycle_us) AND
			NOT Wait
			THEN
			Wait := TRUE;
			gVisionNettime.DAT.NettimeNext_us	:= NettimeCurrent_us + TriggerTimeDelta_us;
			gVisionNettime.DAT.NettimeDelta_us	:= TriggerTimeDelta_us;
			// Transfer nettime to sensor and fire trigger
			IF gVisionSensor[visSelectedSensor].HW.Ready AND NOT gVisionSensor[visSelectedSensor].DAT.ImageProcessingActive THEN
				gVisionSensor[visSelectedSensor].CMD.ImageTrigger	:= TRUE;
				gVisionSensor[visSelectedSensor].DAT.NettimeDelay	:= gVisionNettime.DAT.NettimeNext_us;
			ELSE
				gVisionNettime.DAT.Overflow := gVisionNettime.DAT.Overflow + 1;
			END_IF
			TON_Wait.IN := TRUE;
		END_IF
	END_IF
	TON_Wait(PT := T#1s);
	IF TON_Wait.Q THEN
		TON_Wait.IN := FALSE;
		Wait := FALSE;
	END_IF

//	IF visionResults[0] = 52 THEN
//		visionResultString := 'Shuttle 1';
//	ELSIF visionResults[0] = 51 THEN
//		visionResultString := 'Shuttle 2';
//	ELSIF visionResults[0] = 50 THEN
//		visionResultString := 'Shuttle 3';
//	ELSIF visionResults[0] = 49 THEN
//		visionResultString := 'Shuttle 4';
	//	END_IF

	IF gVisionSensor[3].DAT.ImageNettime <> oldImageNettime THEN
		oldImageNettime := gVisionSensor[3].DAT.ImageNettime;
		brdkStrMemCpy(ADR(visionResultString),ADR(visionResults),SIZEOF(visionResults));
		mappView.updateImage := TRUE;
	END_IF

	mappView.imageFormat 	:= BRDKVIIMG_IMG_TYPE_JPEG;
	mappView.jpegQuality 	:= 50;
	mappView.pSvgImage 		:= ADR(imageSvg);
	//mappView.pImageArray 	:= ADR(this.imgArr);
	//mappView.simulateConfig.activate := DiagCpuIsSimulated(); // true if PLC is simulated
	mappView();

END_PROGRAM

PROGRAM _EXIT
	mappView(enable := FALSE);

END_PROGRAM
```

### Variables.var
```iecst
VAR CONSTANT
	NR_OF_SEGMENTS : USINT := 49; (*50(0..49)*)
END_VAR
VAR
	showMotorSegments : STRING[2000];
	lightValueOld : USINT;
	lightValue : USINT;
END_VAR
VAR RETAIN
	controlLight : lightControlCenter_typ;
END_VAR
```

### Program Logical/Modules/Services/HMI/HMI

#### Types.typ
```iecst
TYPE
	workStationList_typ : 	STRUCT
		listProvider : STRING[800];
		stationCounter : USINT;
		tmpString : STRING[80];
	END_STRUCT;
	local_typ : 	STRUCT
		workStationList : workStationList_typ;
		tableConfigClick : BOOL;
		tableConfigString : STRING[80];
		tableConfigID : USINT;
	END_STRUCT;
	motorSegmentsTyp : 	STRUCT
		visible : BOOL := TRUE;
		ID : STRING[80];
	END_STRUCT;
END_TYPE
```

#### Variables.var
```iecst
VAR
	yCordinate : INT;
	xCordinate : INT;
	i : USINT;
	this : local_typ;
	nrOfShuttlesHMI : USINT := 4;
	pShuttleInfo : REFERENCE TO ShuttleInfoType;
	showConfigShuttles : STRING[5000];
	showShuttles : STRING[5000];
	tmpCalc : REAL;
	tmpString : STRING[5000];
	sizeOfArray : DINT;
	showTyleSvg : BOOL;
	showConfigSvg : BOOL := TRUE;
	showConfigSvgCmd : BOOL;
	showTyleSvgCmd : BOOL;
	gSegments : ARRAY[0..NR_OF_SEGMENTS] OF motorSegmentsTyp;
	pSegments : REFERENCE TO motorSegmentsTyp;
	shuttleStartPosSvgCmd : BOOL;
	shuttleStartPosSvg : BOOL;
	pShuttleStartupInfo : REFERENCE TO shuttleStartup_typ;
	init : BOOL;
	resetMotorSegmentLayoutCmd : BOOL;
	resetShuttleInitLayoutCmd : BOOL;
	lightOutputs : ARRAY[0..5] OF BOOL;
	lightTON : TON;
	currentHMIPage : STRING[80];
END_VAR
```

#### drawMotorSegments.st
```iecst
ACTION drawMotorSegments:
	//manual shuttle config

	IF showTyleSvg OR init THEN
		IF i = 0 THEN
			showMotorSegments := '';
			brdkStrCat(ADR(showMotorSegments), ADR('[{"select":"#MS'));
		ELSE
			brdkStrCat(ADR(showMotorSegments), ADR('{"select":"#MS'));
		END_IF

		tmpString := USINT_TO_STRING(i+1);
		brdkStrCat(ADR(showMotorSegments), ADR(tmpString));
		brdkStrCat(ADR(showMotorSegments), ADR('","display":'));
		IF pSegments.visible THEN
			brdkStrCat(ADR(showMotorSegments), ADR('true'));
		ELSE
			brdkStrCat(ADR(showMotorSegments), ADR('false'));
		END_IF

		IF i = NR_OF_SEGMENTS THEN
			brdkStrCat(ADR(showMotorSegments), ADR('}]'));
		ELSE
			brdkStrCat(ADR(showMotorSegments), ADR('},'));
		END_IF
	END_IF

END_ACTION
```

#### drawShuttles.st
```iecst
ACTION drawShuttles:
	IF i = 0 THEN
		showShuttles := '';
		tmpString := showMotorSegments;
		brdkStrRemove(ADR(tmpString),-1,1);
		brdkStrCat(ADR(showShuttles), ADR(tmpString));
		brdkStrCat(ADR(showShuttles), ADR(','));
	END_IF

	brdkStrCat(ADR(showShuttles), ADR('{"select":"#rect'));

	tmpString := USINT_TO_STRING(i+1);
	brdkStrCat(ADR(showShuttles), ADR(tmpString));
	brdkStrCat(ADR(showShuttles), ADR('","display":'));
	IF (nrOfShuttlesHMI >= (i+1)) THEN
		brdkStrCat(ADR(showShuttles), ADR('true'));
	ELSE
		brdkStrCat(ADR(showShuttles), ADR('false'));
	END_IF

	IF pShuttleInfo.State = mcACP6D_SH_STATE_DISABLED THEN
		brdkStrCat(ADR(showShuttles), ADR(',"fill":3'));
	ELSE
		brdkStrCat(ADR(showShuttles), ADR(',"fill":4'));
	END_IF

	IF pShuttleInfo.State = mcACP6D_SH_STATE_LANDED THEN
		brdkStrCat(ADR(showShuttles), ADR(',"fill":2'));
	ELSE
		brdkStrCat(ADR(showShuttles), ADR(',"fill":4'));
	END_IF

	brdkStrCat(ADR(showShuttles), ADR(',"translate":['));

	tmpCalc := (pShuttleInfo.Position.X*1000)-60;
	tmpString := REAL_TO_STRING(tmpCalc);
	brdkStrCat(ADR(showShuttles), ADR(tmpString));
	brdkStrCat(ADR(showShuttles), ADR(','));

	tmpCalc := 1200 - (pShuttleInfo.Position.Y*1000) - 60;
	tmpString := REAL_TO_STRING(tmpCalc);
	brdkStrCat(ADR(showShuttles), ADR(tmpString));

	IF i = NUM_SHUTTLES THEN
		brdkStrCat(ADR(showShuttles), ADR(']}]'));
	ELSE
		brdkStrCat(ADR(showShuttles), ADR(']},'));
	END_IF

	sizeOfArray := brdkStrLen(ADR(showShuttles));

	//showShuttles := '';
	//showShuttles := '[{"select":"#rect1","display":false, "translate":[100,100]}]';
END_ACTION
```

### Program Logical/Modules/Services/HMI/Vision/Vision (IEC)

#### Main.st - Init, cyclic, exit code
```iecst
PROGRAM _INIT

	//	gVisionNettime.CMD.Activate					:= TRUE;
	//	gVisionNettime.CFG.AxisPeriod				:= 360; // Needs also to be set in the axis configuration
	//	gVisionNettime.CFG.AxisPositionTrigger		:= 0.180;
	//	gVisionNettime.CFG.AxisPositionDelay_Cycles	:= 1; 	// Number of PLK cycles which the axis position is old when it comes to this task (Time from encoder to now in this task)
	//	gVisionNettime.CFG.VisionPreTrigger_Cycles	:= 8; 	// Number of powerlink cycles the trigger has to be send ahead, 4 is a good value.

	mappView.maxSvgImageLength := SIZEOF(imageSvg);
	mappView.enable 		:= TRUE;
	mappView.cameraIp 		:= '192.168.200.8';
	mappView.getImageArray := FALSE;
	mappView.timeout 		:= 3000;

	mappView();

	//TON_Wait.PT := REAL_TO_TIME(154.92);
	TON_Wait.PT := REAL_TO_TIME(3000);

END_PROGRAM

PROGRAM _CYCLIC

	////// Vision sensor configuration /////
	// Must apparently be set in _CYCLIC

	gVisionImage.CFG.EthDevice								:= 'IF2';			// Ethernet interface for the PLC, this is the IF where you go online

	// Configuration for blob
	gVisionSensor[visSelectedSensor].CFG.VisionFunction		:= enumBlob;		// Used to run specific code for this vision function
	gVisionSensor[visSelectedSensor].CFG.PowerlinkNode		:= 8;				// Powerlink node number
	gVisionSensor[visSelectedSensor].CFG.DataStructure		:= ADR(gBlob);		// Global structures that holds all data related to this function
	gVisionSensor[visSelectedSensor].CFG.ComponentLink		:= gCamera;			// Vision component name defined under mappVision in the configuration view
	//gVisionSensor[visSelectedSensor].CFG.ResolutionWidth_X	:= 1280;
	//gVisionSensor[visSelectedSensor].CFG.ResolutionHeight_Y	:= 1024;

	// Camera configuration
	gVisionSensor[visSelectedSensor].FCT.ApplicationName	:= 'ViApplication';
	gVisionSensor[visSelectedSensor].DAT.Exposure			:= 1000; 	// SUSCEPTIBLE TO CHANGE
	gVisionSensor[visSelectedSensor].DAT.FlashColor			:= 4; 		// 4: LIME (See help function "Image acquisition parameters (cyclic write)" for other alternatives)
	gVisionSensor[visSelectedSensor].DAT.FlashSegment		:= 15; 		// Binary 1111 (all segments are turned on)
	gVisionSensor[visSelectedSensor].DAT.Focus				:= 600; 	// SUSCEPTIBLE TO CHANGE - Camera FocusScale is defined in mm
	gVisionSensor[visSelectedSensor].DAT.Gain				:= 1; 								// Gain factor 1
	//gVisionSensor[visSelectedSensor].DAT.MaxItemCnt		:= RecipeData.Cam[i].MaxItemCnt; 	// Already has default value
	//gVisionSensor[visSelectedSensor].DAT.Timeout			:= RecipeData.Cam[i].Timeout; 		// Already has default value

	////////////////////////////////////////

	PowerlinkCycle_us			:= NettimeCurrent_us - NettimeLastCycle_us;
	NettimeLastCycle_us			:= NettimeCurrent_us;

	IF gVisionNettime.CMD.Activate THEN
		//AxisPositionNow			:= ShuttleYPos_m + (-1* ShuttleYSpeed_ms) * PowerlinkCycle_us * gVisionNettime.CFG.AxisPositionDelay_Cycles / 1000000; // When the MpAxis gives us the read position, it is old. So calculate the "now" position
		//TriggerPosDelta			:= gVisionNettime.CFG.AxisPositionTrigger - AxisPositionNow;
		//TriggerTimeDelta_us		:= LREAL_TO_DINT((TriggerPosDelta / ShuttleYSpeed_ms) * 1000000);
		TON_Wait.IN := TRUE;
		// Wait for the moment that axis is in the send trigger window depend on delay by topology and the actual powerlink cycle
		IF TON_Wait.Q THEN
			TON_Wait.IN := FALSE;
			//gVisionNettime.DAT.NettimeNext_us	:= NettimeCurrent_us + TriggerTimeDelta_us;
			//gVisionNettime.DAT.NettimeDelta_us	:= TriggerTimeDelta_us;
			// Transfer nettime to sensor and fire trigger
			IF gVisionSensor[visSelectedSensor].HW.Ready AND NOT gVisionSensor[visSelectedSensor].DAT.ImageProcessingActive THEN
				gVisionSensor[visSelectedSensor].CMD.ImageTrigger	:= TRUE;

				gVisionSensor[visSelectedSensor].DAT.NettimeDelay	:= 0;
			ELSE
				//gVisionNettime.DAT.Overflow := gVisionNettime.DAT.Overflow + 1;
			END_IF
		END_IF
	END_IF

	IF gVisionSensor[visSelectedSensor].DAT.ImageNettime <> oldImageNettime THEN
		oldImageNettime := gVisionSensor[visSelectedSensor].DAT.ImageNettime;
		brdkStrMemCpy(ADR(visionResultString),ADR(visionResults),SIZEOF(visionResults));
		mappView.updateImage := TRUE;
	END_IF

	mappView.imageFormat 	:= BRDKVIIMG_IMG_TYPE_JPEG;
	mappView.jpegQuality 	:= 50;
	mappView.pSvgImage 		:= ADR(imageSvg);
	//mappView.pImageArray 	:= ADR(this.imgArr);
	//mappView.simulateConfig.activate := DiagCpuIsSimulated(); // true if PLC is simulated
	mappView();
	TON_Wait();

END_PROGRAM

PROGRAM _EXIT
	mappView(enable := FALSE);

END_PROGRAM
```

#### Types.typ - Local data types
```iecst
TYPE
	CodeReader_typ : 	STRUCT
		NumberSearch : USINT := 1;
		enableRobustness : BOOL := TRUE;
		codeType : USINT := 7;
		enable : BOOL := TRUE;
	END_STRUCT;
	BlobOutput_typ : 	STRUCT
		enable : BOOL := TRUE;
		numSearchMax : USINT := 1;
		offsetROIX : DINT := 0;
		offsetROIY : DINT := 0;
	END_STRUCT;
	BlobInput_typ : 	STRUCT
		numResults : USINT;
		functionProcessingTime : UINT;
		modelNumber : USINT;
		meanGrayValue : USINT;
		area : UDINT;
		rectangularity : USINT;
		positionX : DINT;
		positionY : DINT;
	END_STRUCT;
END_TYPE
```

#### Variables.var - Local variables
```iecst
VAR
	PowerlinkCycle_us : DINT; (*Powerlink cycletime in microseconds*)
	NettimeLastCycle_us : DINT; (*Old nettime used to calculate Powerlink cycle time*)
	AxisPositionNow : LREAL; (*Calculated positon of the axis position, acopos and network delay times are compensated*)
	TriggerTimeDelta_us : DINT; (*Delta time in microseconds to the next trigger*)
	TriggerPosDelta : LREAL; (*Delta position in units to the next trigger*)
	ShuttleYSpeed_ms : LREAL;
END_VAR
VAR CONSTANT
	LAST_IDX_SH_POS_OLD : USINT := 9;
END_VAR
VAR
	ShuttleYPosOld_m : ARRAY[0..LAST_IDX_SH_POS_OLD] OF LREAL;
	TON_Wait : TON;
	visionResults : ARRAY[0..254] OF USINT;
	visionResultString : STRING[255];
	blobOutput : BlobOutput_typ;
	blobInput : BlobInput_typ;
	mappView : brdkViImg_mappView;
	imageSvg : STRING[6000000];
	oldImageNettime : DINT;
END_VAR
```

### VisionTypes.typ
```iecst
(*-----------------------------------------------------------------------------------------------------------------------------------------*)
(*General vision structures*)

TYPE
	typVisionMain : 	STRUCT
		CMD : typVisionCommand;
		CFG : typVisionConfig;
		DAT : typVisionData;
		FCT : typVisionFunction;
		DIA : typVisionDiag;
		HW : typVisionHW;
	END_STRUCT;
	typVisionCommand : 	STRUCT
		ImageTrigger : BOOL;
		ImageTriggerReset : BOOL;
		AutoSetupStartStop : BOOL;
		VaSwitchApplication : BOOL;
		SaveDiagData : BOOL;
	END_STRUCT;
	typVisionConfig : 	STRUCT
		VisionFunction : enumVisionFunction;
		PowerlinkNode : USINT;
		DataStructure : UDINT;
		ComponentLink : ViComponentType;
	END_STRUCT;
	typVisionFunction : 	STRUCT
		ApplicationName : STRING[40];
		Status : DINT;
	END_STRUCT;
	typVisionDiag : 	STRUCT
		DiagName : STRING[80] := 'diag.tgz';
		Status : DINT;
	END_STRUCT;
	typVisionData : 	STRUCT
		Enable : BOOL := FALSE;
		MaxItemCnt : USINT := 10;
		NettimeDelay : DINT;
		Timeout : UINT := 5000;
		Gain : USINT;
		Focus : UINT;
		Exposure : UDINT;
		FlashColor : USINT := 1;
		FlashSegment : USINT := 15;
		LedColor : USINT;
		IRFilter : BOOL;
		OffsetROIX : DINT;
		OffsetROIY : DINT;
		OffsetROIRotationCenterX : DINT;
		OffsetROIRotationCenterY : DINT;
		OffsetROIOrientation : INT;
		ChromaticLock : BOOL;
		Alignment : USINT;
		AutoSetupGain : USINT;
		AutoSetupFocus : UINT;
		AutoSetupExposure : UDINT;
		AcquisitionAcceptedCnt : USINT;
		AcquisitionCompletedCnt : USINT;
		AcquisitionFailedCnt : USINT;
		LightWarningCnt : USINT;
		ImageProcessingError : UINT;
		ImageProcessingActive : BOOL;
		ImageNettime : DINT;
		ProcessingTimeCamera : UINT;
		ProcessingTimeFunction : UINT;
		ResultCnt : USINT;
		CockpitIsActive : BOOL;
		Status : UDINT;
		StatusText : STRING[30];
		Active : BOOL;
	END_STRUCT;
	typVisionHW : 	STRUCT
		Connected : BOOL;
		Ready : BOOL;
		DigitalInput01 : BOOL;
		DigitalOutput01 : BOOL;
		DigitalOutputStatus01 : BOOL;
		DigitalOutput02 : BOOL;
		DigitalOutputStatus02 : BOOL;
		SerialNumber : UDINT;
		ID : UDINT;
		Variant : UDINT;
		Firmware : UDINT;
		Undervoltage : BOOL;
		Temperature : SINT;
	END_STRUCT;
	enumVisionFunction :
		(
		enumFunctionNone,
		enumBlob,
		enumCoderReader,
		enumMatch,
		enumMeasurement,
		enumOCR
		);
END_TYPE

(*-----------------------------------------------------------------------------------------------------------------------------------------*)
(*General Light structures*)

TYPE
	typLightMain : 	STRUCT
		CMD : typLightCommand;
		CFG : typLightConfig;
		DAT : typLightData;
		HW : typLightHW;
	END_STRUCT;
	typLightCommand : 	STRUCT
		FlashTrigger : BOOL;
		FlashTriggerReset : BOOL;
	END_STRUCT;
	typLightConfig : 	STRUCT
		LightType : enumLightType;
		PowerlinkNode : USINT;
	END_STRUCT;
	typLightData : 	STRUCT
		Enable : USINT := 1;
		FlashColor : USINT := 1;
		FlashSegment : UINT := 15;
		Exposure : UDINT := 200;
		SetAngle : UINT;
		Timeout : UINT := 5000;
		NettimeDelay : DINT;
		FlashAcceptedCnt : USINT;
		FlashCompletedCnt : USINT;
		FlashFailedCnt : USINT;
		Status : UDINT;
	END_STRUCT;
	typLightHW : 	STRUCT
		Connected : BOOL;
		Ready : BOOL;
		SerialNumber : UDINT;
		ID : UDINT;
		Variant : UDINT;
		Firmware : UDINT;
		TemperatureLED : SINT;
		TemperatureControllerBoard : SINT;
		WarningCnt : USINT;
	END_STRUCT;
	enumLightType :
		(
		enumLightNone,
		enumBacklight,
		enumLightbar
		);
END_TYPE

(*-----------------------------------------------------------------------------------------------------------------------------------------*)
(*General nettime structures*)

TYPE
	typVisionNettime : 	STRUCT
		CMD : typNettimeCommand;
		CFG : typNettimeConfig;
		DAT : typNettimeData;
	END_STRUCT;
	typNettimeCommand : 	STRUCT
		Activate : BOOL;
	END_STRUCT;
	typNettimeConfig : 	STRUCT
		AxisPeriod : LREAL; (*Units when period repeats*)
		AxisPositionTrigger : LREAL; (*Position in the period where trigger is fired*)
		AxisPositionDelay_Cycles : LREAL; (*Delay in PLK cycles for the read position from drive*)
		VisionPreTrigger_Cycles : DINT; (*Number of powerlink cycles the trigger has to be send ahead*)
	END_STRUCT;
	typNettimeData : 	STRUCT
		NettimeNext_us : DINT; (*Calculated nettime for next trigger*)
		NettimeDelta_us : DINT; (*Difference between current nettime and calculated nettime for the camera trigger*)
		AxisPosition : LREAL; (*Current axis position*)
		AxisVelocity : LREAL; (*Current axis position*)
		AxisInVelocity : BOOL; (*Indicates that the axis is moving at speed*)
		Overflow : DINT; (*Counts up when a trigger could not be set on time*)
	END_STRUCT;
END_TYPE

(*-----------------------------------------------------------------------------------------------------------------------------------------*)
(*Image upload structures*)

TYPE
	typVisionImage : 	STRUCT
		CMD : typVisionImageCommand;
		CFG : typVisionImageConfig;
		DAT : typVisionImageData;
	END_STRUCT;
	typVisionImageCommand : 	STRUCT
		CreateDir : BOOL;
		DeleteDir : BOOL;
		DeleteImage : BOOL;
		Refresh : BOOL;
		DownloadImage : BOOL;
		SaveImageOnPLC : BOOL;
		ResetError : BOOL;
		RefreshCrosshair : BOOL;
	END_STRUCT;
	typVisionImageConfig : 	STRUCT
		FileDevice : STRING[80];
		DirName : STRING[80];
		CameraIP : STRING[80];
		EthDevice : STRING[80];
		ConvertCycles : UDINT;
		Format : USINT; (*0: jpg. 1: bmp*)
		QualityJPG : USINT;
		UploadBmpJpg : BOOL;
		UploadSVG : BOOL;
	END_STRUCT;
	typVisionImageData : 	STRUCT
		Images : ARRAY[0..19]OF STRING[80];
		Status : UINT;
		VisionDisabled : BOOL;
	END_STRUCT;
END_TYPE

(*-----------------------------------------------------------------------------------------------------------------------------------------*)
(*Vision specific structures*)

TYPE
	typCodeReaderMain : 	STRUCT  (*Code reader structures*)
		CodeType : USINT;
		GradingEnable : BOOL;
		RobustnessEnable : BOOL;
		ParameterMode : USINT;
		ParameterOptimization : USINT;
		BarcodeText : ARRAY[1..MAX_NUM_RESULTS]OF STRING[100];
		BarcodeType : ARRAY[1..MAX_NUM_RESULTS]OF USINT;
		PositionX : ARRAY[1..MAX_NUM_RESULTS]OF DINT;
		PositionY : ARRAY[1..MAX_NUM_RESULTS]OF DINT;
		Orientation : ARRAY[1..MAX_NUM_RESULTS]OF INT;
		Grading : ARRAY[1..MAX_NUM_RESULTS]OF SINT;
		EnhancedGrading : ARRAY[1..23]OF USINT;
	END_STRUCT;
	typBlobMain : 	STRUCT  (*Blob function structures*)
		RegionalFeature : BOOL;
		EnhancedBlobInformation : BOOL := FALSE;
		ModelNumber : ARRAY[1..MAX_NUM_RESULTS]OF USINT;
		Clipped : ARRAY[1..MAX_NUM_RESULTS]OF BOOL;
		Area : ARRAY[1..MAX_NUM_RESULTS]OF UDINT;
		PositionX : ARRAY[1..MAX_NUM_RESULTS]OF DINT;
		PositionY : ARRAY[1..MAX_NUM_RESULTS]OF DINT;
		Orientation : ARRAY[1..MAX_NUM_RESULTS]OF INT;
		MeanGrayValue : ARRAY[1..MAX_NUM_RESULTS]OF USINT;
		Length : ARRAY[1..MAX_NUM_RESULTS]OF UDINT;
		Width : ARRAY[1..MAX_NUM_RESULTS]OF UDINT;
	END_STRUCT;
	typMatchMain : 	STRUCT  (*Match function structures*)
		MinScore : USINT := 70;
		MaxOverlap : USINT;
		ModelNumber : ARRAY[1..MAX_NUM_RESULTS]OF USINT;
		Score : ARRAY[1..MAX_NUM_RESULTS]OF USINT;
		PositionX : ARRAY[1..MAX_NUM_RESULTS]OF DINT;
		PositionY : ARRAY[1..MAX_NUM_RESULTS]OF DINT;
		Orientation : ARRAY[1..MAX_NUM_RESULTS]OF INT;
		Scale : ARRAY[1..MAX_NUM_RESULTS]OF USINT;
		RotCenterX : ARRAY[1..MAX_NUM_RESULTS]OF DINT;
		RotCenterY : ARRAY[1..MAX_NUM_RESULTS]OF DINT;
	END_STRUCT;
	typOCRMain : 	STRUCT  (*OCR function structures*)
		ParameterMode : USINT;
		GradingEnable : BOOL;
		Text : ARRAY[1..MAX_NUM_RESULTS]OF STRING[50];
		Grading : ARRAY[1..MAX_NUM_RESULTS]OF USINT;
		PositionX : ARRAY[1..MAX_NUM_RESULTS]OF DINT;
		PositionY : ARRAY[1..MAX_NUM_RESULTS]OF DINT;
		Orientation : ARRAY[1..MAX_NUM_RESULTS]OF INT;
	END_STRUCT;
	typMTMain : 	STRUCT  (*MT function structures*)
		UseResultAsXY : BOOL;
		ParameterMode : USINT;
		Result : ARRAY[1..MAX_NUM_RESULTS]OF DINT;
	END_STRUCT;
END_TYPE

(*------------------------------------------------------------------------------------------------------------------------------------------------------------------------------------------------------------------------*)
(*Structure that contains the recipe variables*)

TYPE
	recVariable : 	STRUCT
		Cam : ARRAY[1..MAX_NUM_CAMS]OF recVariableCam;
		Light : ARRAY[1..MAX_NUM_LIGHTS]OF recVariableLight;
	END_STRUCT;
	recVariableCam : 	STRUCT
		ApplicationName : STRING[40];
		MaxItemCnt : USINT := 10;
		Timeout : UINT := 5000;
		Gain : USINT;
		Focus : UINT;
		Exposure : UDINT;
		FlashColor : USINT := 1;
		FlashSegment : USINT := 15;
	END_STRUCT;
	recVariableLight : 	STRUCT
		Timeout : UINT := 5000;
		Exposure : UDINT;
		FlashColor : USINT := 1;
		FlashSegment : UINT := 15;
		SetAngle : UINT := 45;
	END_STRUCT;
END_TYPE
```

### VisionVariables.var
```iecst
(*-----------------------------------------------------------------------------------------------------------------------------------------*)
(*Global variables for sensor hardware and vision functions*)
VAR
	gBlob : typBlobMain; (*Data that is specific for the blob function*)
	gCodeReader : typCodeReaderMain; (*Data that is specific for the code reader*)
	gMatch : typMatchMain; (*Data that is specific for the match function*)
	gMT : typMTMain; (*Data that is specific for the measurement function*)
	gOCR : typOCRMain; (*Data that is specific for the OCR function*)
	gVisionImage : typVisionImage; (*Data for image handling*)
	gVisionLight : ARRAY[1..MAX_NUM_LIGHTS] OF typLightMain; (*General Light  functions that are independent from the inspection function*)
	gVisionNettime : typVisionNettime; (*Data for nettime calculation*)
	gVisionSensor : ARRAY[1..MAX_NUM_CAMS] OF typVisionMain; (*General vision functions that are independent from the inspection function*)
	NettimeCurrent_us : DINT; (*Current Powerlink nettime*)
	visSelectedSensor : UINT := 3; (*Selected camera node number*)
	visSelectedLight : UINT := 1; (*Selected Light node number*)
END_VAR
VAR RETAIN
	RecipeData : recVariable; (*Structure that contains the recipe variables*)
END_VAR
(*-----------------------------------------------------------------------------------------------------------------------------------------*)
(*Global constants*)
VAR CONSTANT
	MAX_NUM_CAMS : UINT := 5; (*Maximum number of camera's*)
	MAX_NUM_LIGHTS : UINT := 5; (*Maximum number of light's*)
	MAX_NUM_RESULTS : UINT := 10; (*Maximum number of results*)
	MAX_IDX_VA_LIST : UINT := 19; (*Maximum number of entrys in the Vision Application list*)
	DEVICE_NAME : STRING[40] := 'VisionFileDevice'; (*File device where the images and recipes are stored*)
	NETTIME_DEFAULT_DELAY : UDINT := 30000; (*This delay is used when software trigger is used and nettime is enabled*)
	MAX_NUM_CODETYPES : USINT := 69; (*Maximum number of code types*)
END_VAR
VAR
	CodeTypes : {REDUND_UNREPLICABLE} ARRAY[0..MAX_NUM_CODETYPES] OF STRING[80] := ['Auto Identify (0)','2/5 Industrial (1)','2/5 Interleaved (2)','Codebar (3)','Code 32 (4)','Code 39 (5)','Code 93 (6)','Code 128 (7)','MSI (8)','PharmaCode (9)','EAN-8 (10)','EAN-8 Add-On 2 (11)','EAN-8 Add-On 5 (12)','EAN-13 (13)','EAN-13 Add-On 2 (14)','EAN-13 Add-On 5 (15)',4(''),'UPC-A (20)','UPC-A Add-On 2 (21)','UPC-A Add-On 5 (22)','UPC-E (23)','UPC-E Add-On 2 (24)','UPC-E Add-On 5 (25)',4(''),'GS1-128 (30)','GS1 DataBar Omnidirectional (31)','GS1 DataBar Truncated (32)','GS1 DataBar Stacked (33)','GS1 DataBar Stacked Omnidirectional (34)','GS1 DataBar Limited (35)','GS1 DataBar Expanded (36)','GS1 DataBar ExpandedStacked (37)',12(''),'Data Matrix ECC200 (50)','QR Code Model 1 (51)','QR Code Model 2 (52)','Micro QRCode (53)','PDF417 (54)','Aztec Code (55)',4(''),'GS1 Data Matrix (60)','GS1 QR Code Model 1 (61)','GS1 QR Code Model 2 (62)','GS1 Aztec Code (63)',6('')];
END_VAR
```

### Program Logical/Modules/Services/HMI/Vision/Vi_main (IEC)

#### Variables.var
```iecst
(*-----------------------------------------------------------------------------------------------------------------------------------------*)
(*Main vision and data structures*)
VAR
	VisionSensor : REFERENCE TO typVisionMain; (*General vision functions that are independent from the inspection function*)
	Match : REFERENCE TO typMatchMain; (*Data that is specific for the match function*)
	CodeReader : REFERENCE TO typCodeReaderMain; (*Data that is specific for the code reader*)
	MT : REFERENCE TO typMTMain; (*Data that is specific for the MT function*)
	OCR : REFERENCE TO typOCRMain; (*Data that is specific for the OCR function*)
	Blob : REFERENCE TO typBlobMain; (*Data that is specific for the blob function*)
	tmpMatch : {REDUND_UNREPLICABLE} typMatchMain; (*Data that is specific for the match function*)
	tmpCodeReader : {REDUND_UNREPLICABLE} typCodeReaderMain; (*Data that is specific for the code reader*)
	tmpMT : {REDUND_UNREPLICABLE} typMTMain; (*Data that is specific for the OCR function*)
	tmpOCR : {REDUND_UNREPLICABLE} typOCRMain; (*Data that is specific for the OCR function*)
	tmpBlob : {REDUND_UNREPLICABLE} typBlobMain; (*Data that is specific for the blob function*)
END_VAR
(*-----------------------------------------------------------------------------------------------------------------------------------------*)
(*Vision function blocks*)
VAR
	VaGetList_01 : VaGetList;
	ViBaseLoadApplication_01 : ViBaseLoadApplication;
	ViBaseSaveDiagData_01 : ViBaseSaveDiagData;
	FDelete : FileDelete;
END_VAR
(*-----------------------------------------------------------------------------------------------------------------------------------------*)
(*Local variables*)
VAR
	idx : UINT;
	visTableNo : ARRAY[1..MAX_NUM_RESULTS] OF USINT := [1,2,3,4,5,6,7,8,9,10];
	visEnableCommand : BOOL; (*Enable/Disable vision trigger and enable when camera is not ready*)
	visEnableSetup : BOOL; (*Enable/Disable vision setup when camera is not ready*)
	visEnableRepetitive : BOOL; (*Enable/Disable repetitive mode*)
	visEnableVision : BOOL; (*Enable vision function*)
	visAutoArchiv : BOOL; (*Enable/Disable auto archiving of camera images*)
	visImageTrigger : BOOL; (*Trigger new image*)
	TriggerTimeout : ARRAY[1..MAX_NUM_CAMS] OF TON; (*Disable web reload when timed out*)
	visVisionApplicationList : ARRAY[0..19] OF STRING[80]; (*Flash color string*)
	visSelectedFlashColor : STRING[10]; (*Flash color string*)
	visSelectedFlashColorOld : STRING[10]; (*Flash color string*)
	visSelectedFlashSegment : ARRAY[0..3] OF USINT := [4(1)]; (*Selected flash segments*)
	visSelectedFlashSegmentOld : ARRAY[0..3] OF USINT := [4(1)]; (*Selected flash segments*)
	visRepetitiveMode : BOOL; (*Enable/Disable repetitive mode*)
	RepetitiveModeTimer : TON; (*Timer for repetitive mode*)
	DisableAutoArchiv : BOOL; (*Enable/Disable automatic archieving for images*)
	AcquisitionFailedCntOld : ARRAY[1..MAX_NUM_CAMS] OF UDINT; (*Old aquisition failed counter*)
	AcquisitionCompletedCntOld : ARRAY[1..MAX_NUM_CAMS] OF UDINT; (*Old aquisition completed counter*)
	InitialSearchSensor : BOOL; (*Flag for first boot*)
	AutoSetupRunning : ARRAY[1..MAX_NUM_CAMS] OF BOOL; (*Flag for auto setup running*)
END_VAR

(*-----------------------------------------------------------------------------------------------------------------------------------------*)
(*Image, crosshair data and constants*)
VAR
	tmpStr1 : STRING[1000];
	i : UINT;
	visCameraStatus : STRING[30];
END_VAR
VAR CONSTANT
	HexTab : STRING[16] := '0123456789ABCDEF';
END_VAR
(*-----------------------------------------------------------------------------------------------------------------------------------------*)
(*Error numbers*)
VAR CONSTANT
	ERR_VA_LIST_NUM : UINT := 30000; (*Number of applications exceeds array size*)
END_VAR
VAR
	TON_DelayAfterAutoSetup : TON;
	visVaListRefresh : BOOL;
END_VAR
```

#### Main.st
```iecst
// --------------------------------------------------------------------------------------------------------------------
// General vision task. This is a support task for the mappView visualization. The following functions are implemneted
// - Disable mappView functions when camera is not ready, available
// - Load image on main page when camera has finished inspection
// - Transfer parameters after vision setup
// - Draw crosshairs into image on the main page
// Version 2.x (Check revision history for details)
// --------------------------------------------------------------------------------------------------------------------
PROGRAM _INIT
	// -----------------------------------------------------------------------------------------------------------
	// Map global structure to local reference
	VisionSensor ACCESS ADR(gVisionSensor[visSelectedSensor]);
	Blob ACCESS ADR(tmpBlob);
	CodeReader ACCESS ADR(tmpCodeReader);
	Match ACCESS ADR(tmpMatch);
	MT ACCESS ADR(tmpMT);
	OCR ACCESS ADR(tmpOCR);

	// -----------------------------------------------------------------------------------------------------------
	visTableNo;
	InitialSearchSensor := TRUE;
END_PROGRAM

// -----------------------------------------------------------------------------------------------------------
// Cyclic part
// -----------------------------------------------------------------------------------------------------------
PROGRAM _CYCLIC
// -----------------------------------------------------------------------------------------------------------
// Part 1: Things to be done for every camera/sensor
// -----------------------------------------------------------------------------------------------------------
	FOR idx := 1 TO MAX_NUM_CAMS DO
		// -----------------------------------------------------------------------------------------------------------
		// Display camera status in hex - documentation is also in hex
		// -----------------------------------------------------------------------------------------------------------
		IF gVisionSensor[idx].DAT.Status = 0 THEN // Display only a single 0
			gVisionSensor[idx].DAT.StatusText := '0';
		ELSIF gVisionSensor[idx].DAT.Status = 16#00000001 THEN
			gVisionSensor[idx].DAT.StatusText := 'Image acquisition';
		ELSIF gVisionSensor[idx].DAT.Status = 16#00000002 THEN
			gVisionSensor[idx].DAT.StatusText := 'Waiting trigger';
		ELSIF gVisionSensor[idx].DAT.Status = 16#00000010 THEN
			gVisionSensor[idx].DAT.StatusText := 'Searching settings';
		ELSIF gVisionSensor[idx].DAT.Status = 16#00000080 THEN
			gVisionSensor[idx].DAT.StatusText := 'Setting focus';
		ELSIF gVisionSensor[idx].DAT.Status = 16#00000090 THEN
			gVisionSensor[idx].DAT.StatusText := 'Searching settings';
		ELSIF gVisionSensor[idx].DAT.Status = 16#00000800 THEN
			gVisionSensor[idx].DAT.StatusText := 'Cam CPU not ready';
		ELSIF gVisionSensor[idx].DAT.Status = 16#00001000 THEN
			gVisionSensor[idx].DAT.StatusText := 'Cam sensor not ready';
		ELSIF gVisionSensor[idx].DAT.Status = 16#02000000 THEN
			gVisionSensor[idx].DAT.StatusText := 'OS check/update';
		ELSIF gVisionSensor[idx].DAT.Status = 16#80000000 THEN
			gVisionSensor[idx].DAT.StatusText := 'Vision cockpit active';
		ELSE // Display the status in hex format 0x02000800
			gVisionSensor[idx].DAT.StatusText := '';
			FOR i := 0 TO 28 BY 4 DO
				gVisionSensor[idx].DAT.StatusText := CONCAT(MID(HexTab, 1, LIMIT(1, UDINT_TO_INT((SHR(gVisionSensor[idx].DAT.Status, i) AND 16#0000000F) + 1), 16)), gVisionSensor[idx].DAT.StatusText);
			END_FOR
			gVisionSensor[idx].DAT.StatusText := CONCAT('0x', gVisionSensor[idx].DAT.StatusText);
		END_IF

		// -----------------------------------------------------------------------------------------------------------
		// Check if vision cockpit is open
		// -----------------------------------------------------------------------------------------------------------
		gVisionSensor[idx].DAT.CockpitIsActive := (gVisionSensor[idx].DAT.Status AND 16#8000_0000) > 0;

		// -----------------------------------------------------------------------------------------------------------
		// Auto setup handling
		// -----------------------------------------------------------------------------------------------------------
		IF(gVisionSensor[idx].CMD.AutoSetupStartStop AND gVisionSensor[idx].DAT.Status <> 0) THEN
			AutoSetupRunning[idx] := TRUE;
		ELSIF NOT gVisionSensor[idx].CMD.AutoSetupStartStop THEN
			AutoSetupRunning[idx] := FALSE;
		END_IF
		IF(gVisionSensor[idx].CMD.AutoSetupStartStop AND gVisionSensor[idx].DAT.Status = 0 AND AutoSetupRunning[idx]) THEN // Setup successfully finished
			gVisionSensor[idx].DAT.Gain					:= gVisionSensor[idx].DAT.AutoSetupGain;
			gVisionSensor[idx].DAT.Focus				:= gVisionSensor[idx].DAT.AutoSetupFocus;
			gVisionSensor[idx].DAT.Exposure				:= gVisionSensor[idx].DAT.AutoSetupExposure;
			gVisionSensor[idx].CMD.AutoSetupStartStop	:= FALSE;
			AutoSetupRunning[idx]						:= FALSE;
			TON_DelayAfterAutoSetup.IN					:= TRUE;
		END_IF
		TON_DelayAfterAutoSetup(PT := T#50ms);
		IF TON_DelayAfterAutoSetup.Q THEN // After the camera tells it is ready, we need to wait still at least ca 20ms, otherwise it does not accept the trigger
			TON_DelayAfterAutoSetup.IN := FALSE;
			IF gVisionSensor[idx].HW.Ready AND NOT gVisionSensor[idx].DAT.ImageProcessingActive THEN
				gVisionSensor[idx].DAT.NettimeDelay	:= NettimeCurrent_us + NETTIME_DEFAULT_DELAY;
				gVisionSensor[idx].CMD.ImageTrigger	:= TRUE;
				gVisionSensor[idx].DAT.Active			:= TRUE;
			END_IF
		END_IF

		// -----------------------------------------------------------------------------------------------------------
		// Reset image trigger, reload web page and store image when process is finished
		// -----------------------------------------------------------------------------------------------------------
		IF ((gVisionSensor[idx].DAT.AcquisitionCompletedCnt <> AcquisitionCompletedCntOld[idx] OR gVisionSensor[idx].DAT.AcquisitionFailedCnt <> AcquisitionFailedCntOld[idx]) AND NOT gVisionSensor[idx].DAT.ImageProcessingActive AND gVisionSensor[idx].HW.Ready) THEN
			AcquisitionCompletedCntOld[idx]			:= gVisionSensor[idx].DAT.AcquisitionCompletedCnt;
			AcquisitionFailedCntOld[idx]			:= gVisionSensor[idx].DAT.AcquisitionFailedCnt;
			gVisionSensor[idx].CMD.ImageTrigger		:= FALSE;
			gVisionSensor[idx].DAT.Active			:= FALSE;
			// Store image to flash card, only for the actual selected camera
			IF idx = visSelectedSensor THEN
				IF visAutoArchiv AND NOT DisableAutoArchiv THEN
					gVisionImage.CMD.SaveImageOnPLC := TRUE;
				END_IF
				IF NOT visRepetitiveMode THEN
					DisableAutoArchiv := FALSE;
				END_IF
			END_IF
		END_IF

		// -----------------------------------------------------------------------------------------------------------
		// Reset trigger when timed out
		// -----------------------------------------------------------------------------------------------------------
		IF gVisionSensor[idx].CMD.ImageTrigger THEN
			TriggerTimeout[idx].IN := TRUE;
			TriggerTimeout[idx].PT := REAL_TO_TIME(gVisionSensor[idx].DAT.Timeout * 1.25);
			IF TriggerTimeout[idx].Q THEN
				gVisionSensor[idx].CMD.ImageTrigger			:= FALSE;
				gVisionSensor[idx].CMD.ImageTriggerReset	:= TRUE;
				gVisionSensor[idx].DAT.Active				:= FALSE;
			END_IF
		ELSE
			TriggerTimeout[idx].IN := FALSE;
			gVisionSensor[idx].CMD.ImageTriggerReset := FALSE;
		END_IF
		TriggerTimeout[idx]();
	END_FOR

// -----------------------------------------------------------------------------------------------------------
// Part 2: Things to be done for the actual selected camera / visualization related things
// -----------------------------------------------------------------------------------------------------------
	// -----------------------------------------------------------------------------------------------------------
	// Select first available camera after reboot
	// -----------------------------------------------------------------------------------------------------------
	IF InitialSearchSensor THEN
		FOR i := 1 TO MAX_NUM_CAMS DO
			IF gVisionSensor[i].HW.Connected THEN
				visSelectedSensor := i;
				InitialSearchSensor := FALSE;
				EXIT;
			END_IF
		END_FOR
		visVaListRefresh := TRUE;
	END_IF

	// -----------------------------------------------------------------------------------------------------------
	// Map global structure to local reference for mappView
	// -----------------------------------------------------------------------------------------------------------
	// Make sure we dont exceed array limit
	IF(visSelectedSensor > MAX_NUM_CAMS) THEN
		visSelectedSensor := 1;
	END_IF
	IF(visSelectedSensor < 1) THEN
		visSelectedSensor := MAX_NUM_CAMS;
	END_IF
	// -----------------------------------------------------------------------------------------------------------
	// Assign pointers
	VisionSensor ACCESS ADR(gVisionSensor[visSelectedSensor]);
	IF(VisionSensor.CFG.DataStructure <> 0) THEN
		CASE VisionSensor.CFG.VisionFunction OF
			enumBlob:			Blob ACCESS VisionSensor.CFG.DataStructure;
			enumCoderReader:	CodeReader ACCESS VisionSensor.CFG.DataStructure;
			enumMatch:			Match ACCESS VisionSensor.CFG.DataStructure;
			enumMeasurement:	MT ACCESS VisionSensor.CFG.DataStructure;
			enumOCR:			OCR ACCESS VisionSensor.CFG.DataStructure;
		END_CASE
	ELSE
		RETURN;
	END_IF

	// -----------------------------------------------------------------------------------------------------------
	// Display camera status
	// -----------------------------------------------------------------------------------------------------------
	visCameraStatus := VisionSensor.DAT.StatusText;

	// -----------------------------------------------------------------------------------------------------------
	// Camera with blob function
	// -----------------------------------------------------------------------------------------------------------
	IF VisionSensor.CFG.VisionFunction = enumBlob THEN
		//Do some processing
	END_IF

	// -----------------------------------------------------------------------------------------------------------
	// Translate flash color and segments from mappView to IO mapping
	// -----------------------------------------------------------------------------------------------------------
	// Hint: Normally copy from recipe (VisionSensor) to visu. Only in case of a change in the visu copy to recipe
	IF visSelectedFlashColor <> visSelectedFlashColorOld THEN // The flash color was changed in the mappView visualization
		VisionSensor.DAT.FlashColor := UDINT_TO_USINT(brsatoi(ADR(visSelectedFlashColor)));
	ELSE
		brsitoa(VisionSensor.DAT.FlashColor, ADR(visSelectedFlashColor));
	END_IF
	visSelectedFlashColorOld := visSelectedFlashColor;
	IF brsmemcmp(ADR(visSelectedFlashSegment), ADR(visSelectedFlashSegmentOld), SIZEOF(visSelectedFlashSegment)) <> 0 THEN // The flash segments was changed in the mappView visualization
		VisionSensor.DAT.FlashSegment := SHL(visSelectedFlashSegment[0], 0) OR SHL(visSelectedFlashSegment[1], 1) OR SHL(visSelectedFlashSegment[2], 2) OR SHL(visSelectedFlashSegment[3], 3);
	ELSE
		visSelectedFlashSegment[0] := VisionSensor.DAT.FlashSegment.0;
		visSelectedFlashSegment[1] := VisionSensor.DAT.FlashSegment.1;
		visSelectedFlashSegment[2] := VisionSensor.DAT.FlashSegment.2;
		visSelectedFlashSegment[3] := VisionSensor.DAT.FlashSegment.3;
	END_IF
	visSelectedFlashSegmentOld := visSelectedFlashSegment;

	// -----------------------------------------------------------------------------------------------------------
	// Disable command buttons when camera is disconnected, not ready, processing an image or vision cockpit is open
	// -----------------------------------------------------------------------------------------------------------
	IF(NOT VisionSensor.HW.Connected OR NOT VisionSensor.HW.Ready OR VisionSensor.DAT.ImageProcessingActive OR VisionSensor.DAT.CockpitIsActive) THEN
		visEnableCommand := FALSE;
	ELSE
		visEnableCommand := TRUE;
	END_IF

	// -----------------------------------------------------------------------------------------------------------
	// Disable setup buttons when camera is disconnected, processing an image or not ready
	// -----------------------------------------------------------------------------------------------------------
	IF(NOT VisionSensor.HW.Connected OR NOT (VisionSensor.HW.Ready OR AutoSetupRunning[visSelectedSensor]) OR VisionSensor.DAT.ImageProcessingActive) THEN
		visEnableSetup := FALSE;
	ELSE
		visEnableSetup := TRUE;
	END_IF

	// -----------------------------------------------------------------------------------------------------------
	// Fire trigger for camera image
	// -----------------------------------------------------------------------------------------------------------
	IF((visImageTrigger OR EDGEPOS(visEnableVision)) AND VisionSensor.HW.Ready AND NOT VisionSensor.DAT.ImageProcessingActive) THEN
		// Add default delay and fire trigger
		VisionSensor.DAT.NettimeDelay	:= NettimeCurrent_us + NETTIME_DEFAULT_DELAY;
		VisionSensor.CMD.ImageTrigger	:= TRUE;
		visImageTrigger					:= FALSE;
		VisionSensor.DAT.Active			:= TRUE;
	END_IF

	// -----------------------------------------------------------------------------------------------------------
	// Repetitive mode
	// -----------------------------------------------------------------------------------------------------------
	visEnableRepetitive := visEnableCommand OR visRepetitiveMode; // Enable of the repetitive mode button. Don't disable while repetitive mode is active
	IF visRepetitiveMode THEN
		RepetitiveModeTimer.IN := TRUE;
		IF RepetitiveModeTimer.Q THEN
			IF VisionSensor.HW.Ready AND NOT VisionSensor.DAT.ImageProcessingActive THEN
				RepetitiveModeTimer.IN := FALSE;
				VisionSensor.DAT.NettimeDelay := NettimeCurrent_us + NETTIME_DEFAULT_DELAY;
				VisionSensor.CMD.ImageTrigger := TRUE;
			END_IF
		END_IF
		DisableAutoArchiv := TRUE;
	ELSE
		RepetitiveModeTimer.IN := TRUE;
	END_IF
	RepetitiveModeTimer(PT := T#200ms);
	VisionSensor.DAT.Enable := visEnableVision AND NOT visRepetitiveMode;

	// -----------------------------------------------------------------------------------------------------------
	// Get list of vision applications and components
	// -----------------------------------------------------------------------------------------------------------
	IF (visVaListRefresh) THEN
		VaGetList_01(Enable := TRUE);
		VisionSensor.FCT.Status := ERR_FUB_BUSY;
		IF VaGetList_01.Status <> ERR_FUB_BUSY THEN
			// Convert vision application list to mappView format
			IF VaGetList_01.Status = ERR_OK THEN
				IF VaGetList_01.VaApplicationCnt > 0 AND VaGetList_01.VaApplicationCnt < MAX_IDX_VA_LIST THEN
					FOR i:=0 TO VaGetList_01.VaApplicationCnt - 1 DO
						String2DataProvider(ADR(VaGetList_01.VaApplicationNames[i]), ADR(visVisionApplicationList[i]));
					END_FOR
				END_IF
				VisionSensor.FCT.Status := ERR_OK;
			ELSE // Error
				brsmemset(ADR(visVisionApplicationList), 0, SIZEOF(visVisionApplicationList));
				VisionSensor.FCT.Status := VaGetList_01.Status;
			END_IF
			// Reset function block
			VaGetList_01(Enable := FALSE);
			visVaListRefresh := FALSE;
		END_IF
	END_IF

	// -----------------------------------------------------------------------------------------------------------
	// Load vision application
	// -----------------------------------------------------------------------------------------------------------
	IF (VisionSensor.CMD.VaSwitchApplication) THEN
		ViBaseLoadApplication_01.MpLink	:= ADR(VisionSensor.CFG.ComponentLink);
		ViBaseLoadApplication_01.Name	:= ADR(VisionSensor.FCT.ApplicationName);
		VisionSensor.FCT.Status := ERR_FUB_BUSY;

		// -----------------------------------------------------------------------------------------------------------
		// OK
		IF (ViBaseLoadApplication_01.Done) THEN
			VisionSensor.FCT.Status := ERR_OK;
			VisionSensor.CMD.VaSwitchApplication := FALSE;
		// -----------------------------------------------------------------------------------------------------------
		// Error
		ELSIF (NOT ViBaseLoadApplication_01.Busy AND ViBaseLoadApplication_01.Error) THEN
			VisionSensor.FCT.Status := ViBaseLoadApplication_01.StatusID;
			VisionSensor.CMD.VaSwitchApplication := FALSE;
		END_IF
	END_IF
	ViBaseLoadApplication_01.Execute := VisionSensor.CMD.VaSwitchApplication;
	ViBaseLoadApplication_01();

	// -----------------------------------------------------------------------------------------------------------
	// Informations for Vi_image
	// -----------------------------------------------------------------------------------------------------------
	IF EDGENEG(VisionSensor.DAT.ImageProcessingActive) THEN
		gVisionImage.CMD.RefreshCrosshair := TRUE;
	END_IF
	gVisionImage.DAT.VisionDisabled := NOT visEnableVision;

	// -----------------------------------------------------------------------------------------------------------
	// Save diagnostic data
	// -----------------------------------------------------------------------------------------------------------
	IF (VisionSensor.CMD.SaveDiagData) THEN
		// Delete old file first
		FDelete.enable := VisionSensor.CMD.SaveDiagData AND NOT ViBaseSaveDiagData_01.Execute;
		FDelete.pDevice := ADR(DEVICE_NAME);
		FDelete.pName := ADR(VisionSensor.DIA.DiagName);
		IF (FDelete.status <> ERR_FUB_BUSY) THEN
			ViBaseSaveDiagData_01.Execute := TRUE;
		END_IF
		// Upload diagnostic information
		ViBaseSaveDiagData_01.MpLink := ADR(VisionSensor.CFG.ComponentLink);
		ViBaseSaveDiagData_01.DeviceName := ADR(DEVICE_NAME);
		ViBaseSaveDiagData_01.FileName := ADR(VisionSensor.DIA.DiagName);
		VisionSensor.DIA.Status := ERR_FUB_BUSY;

		// -----------------------------------------------------------------------------------------------------------
		// OK
		IF (ViBaseSaveDiagData_01.Done) THEN
			VisionSensor.DIA.Status := ERR_OK;
			ViBaseSaveDiagData_01.Execute := FALSE;
			VisionSensor.CMD.SaveDiagData := FALSE;
		// -----------------------------------------------------------------------------------------------------------
		// Error
		ELSIF (NOT ViBaseSaveDiagData_01.Busy AND ViBaseSaveDiagData_01.Error) THEN
			VisionSensor.DIA.Status := ViBaseSaveDiagData_01.StatusID;
			ViBaseSaveDiagData_01.Execute := FALSE;
			VisionSensor.CMD.SaveDiagData := FALSE;
		END_IF
	END_IF
	ViBaseSaveDiagData_01();
	FDelete();

END_PROGRAM
```

- Visualisation Logical/mappView (not shown)

Listed in the project but not available here: Logical/Global.typ, Logical/Modules/Main/Variables.var, Logical/Modules/Acopos6D/Acopos6D/shuttleGroups.st, Logical/Modules/Acopos6D/Acopos6D/WeightProgram.st, Logical/Modules/Acopos6D/Acopos6D/MovementRxRyRz.st, Logical/Modules/Acopos6D/Acopos6D/AreWorkstations.st, Logical/Modules/KUKA/CTRL/mxA_ErrorMessage.st, Logical/Modules/KUKA/CTRL/mxA_JointMovement.st, Logical/Modules/KUKA/CTRL/LocalFunctions.fun, Logical/Modules/KUKA/CTRL/GripperAction.st, Logical/Modules/KUKA/KUKA/GripperAction.st, Logical/Modules/KUKA/Services/HMI/Variables.var
